LIN {X 0,Y 288.913,Z 1256.965,A -85,B 0,C 180,E1 22492.445,E2 22492.445} C_VEL
LIN {X 0,Y 288.678,Z 1266.037,A -85,B 0,C 180,E1 22499.979,E2 22499.979} C_VEL
LIN {X 0,Y 289.252,Z 1269.357,A -85,B 0,C 180,E1 22505.992,E2 22505.992} C_VEL
LIN {X 0,Y 291.406,Z 1269.606,A -85,B 0,C 180,E1 22511.982,E2 22511.982} C_VEL
LIN {X 0,Y 298.511,Z 1264.594,A -85,B 0,C 180,E1 22520.789,E2 22520.789} C_VEL
LIN {X 0,Y 311.662,Z 1253.252,A -85,B 0,C 180,E1 22529.064,E2 22529.064} C_VEL
LIN {X 0,Y 331.336,Z 1236.016,A -85,B 0,C 180,E1 22536.45,E2 22536.45} C_VEL
LIN {X 0,Y 358.761,Z 1211.96,A -85,B 0,C 180,E1 22542.945,E2 22542.945} C_VEL
LIN {X 0,Y 361.98,Z 1209.227,A -85,B 0,C 180,E1 22543.828,E2 22543.828} C_VEL
LIN {X 0,Y 332.745,Z 1238.454,A -85,B 0,C 180,E1 22549.983,E2 22549.983} C_VEL
LIN {X 0,Y 312.443,Z 1260.562,A -85,B 0,C 180,E1 22556.95,E2 22556.95} C_VEL
LIN {X 0,Y 299.017,Z 1276.755,A -85,B 0,C 180,E1 22564.501,E2 22564.501} C_VEL
LIN {X 0,Y 291.853,Z 1286.905,A -85,B 0,C 180,E1 22571.864,E2 22571.864} C_VEL
LIN {X 0,Y 289.278,Z 1291.684,A -85,B 0,C 180,E1 22577.92,E2 22577.92} C_VEL
LIN {X 0,Y 288.568,Z 1293.172,A -85,B 0,C 180,E1 22585.704,E2 22585.704} C_VEL
LIN {X 0,Y 288.992,Z 1290.468,A -85,B 0,C 180,E1 22591.516,E2 22591.516} C_VEL
LIN {X 0,Y 289.159,Z 1283.794,A -85,B 0,C 180,E1 22597.542,E2 22597.542} C_VEL
LIN {X 0,Y 290.047,Z 1270.937,A -85,B 0,C 180,E1 22604.382,E2 22604.382} C_VEL
LIN {X 0,Y 290.956,Z 1264.711,A -85,B 0,C 180,E1 22607.439,E2 22607.439} C_VEL
LIN {X 0,Y 296.193,Z 1251.831,A -85,B 0,C 180,E1 22614.979,E2 22614.979} C_VEL
LIN {X 0,Y 306.956,Z 1232.131,A -85,B 0,C 180,E1 22622.484,E2 22622.484} C_VEL
LIN {X 0,Y 322.211,Z 1206.964,A -85,B 0,C 180,E1 22628.94,E2 22628.94} C_VEL
LIN {X 0,Y 340.045,Z 1177.266,A -85,B 0,C 180,E1 22634.144,E2 22634.144} C_VEL
LIN {X 0,Y 358.723,Z 1143.523,A -85,B 0,C 180,E1 22638.132,E2 22638.132} C_VEL
LIN {X 0,Y 372.662,Z 1114.646,A -85,B 0,C 180,E1 22640.6,E2 22640.6} C_VEL
LIN {X 0,Y 373.421,Z 1108.193,A -85,B 0,C 180,E1 22642.533,E2 22642.533} C_VEL
LIN {X 0,Y 372.674,Z 1104.982,A -85,B 0,C 180,E1 22645.328,E2 22645.328} C_VEL
LIN {X 0,Y 372.153,Z 1105.867,A -85,B 0,C 180,E1 22648.785,E2 22648.785} C_VEL
LIN {X 0,Y 371.814,Z 1111.068,A -85,B 0,C 180,E1 22651.664,E2 22651.664} C_VEL
LIN {X 0,Y 356.252,Z 1142.151,A -85,B 0,C 180,E1 22654.514,E2 22654.514} C_VEL
LIN {X 0,Y 340.752,Z 1167.55,A -85,B 0,C 180,E1 22658.157,E2 22658.157} C_VEL
LIN {X 0,Y 330.737,Z 1181.649,A -85,B 0,C 180,E1 22661.066,E2 22661.066} C_VEL
LIN {X 0,Y 320.798,Z 1191.408,A -85,B 0,C 180,E1 22662.97,E2 22662.97} C_VEL
LIN {X 0,Y 312.043,Z 1198.825,A -85,B 0,C 180,E1 22664.79,E2 22664.79} C_VEL
LIN {X 0,Y 311.157,Z 1199.698,A -85,B 0,C 180,E1 22665.117,E2 22665.117} C_VEL
LIN {X 0,Y 298.817,Z 1210.613,A -85,B 0,C 180,E1 22671.272,E2 22671.272} C_VEL
LIN {X 0,Y 291.006,Z 1214.857,A -85,B 0,C 180,E1 22677.037,E2 22677.037} C_VEL
LIN {X 0,Y 285.807,Z 1214.307,A -85,B 0,C 180,E1 22683.06,E2 22683.06} C_VEL
LIN {X 0,Y 283.385,Z 1208.666,A -85,B 0,C 180,E1 22689.252,E2 22689.252} C_VEL
LIN {X 0,Y 283.421,Z 1196.875,A -85,B 0,C 180,E1 22695.723,E2 22695.723} C_VEL
LIN {X 0,Y 285.142,Z 1180.307,A -85,B 0,C 180,E1 22701.438,E2 22701.438} C_VEL
LIN {X 0,Y 288.359,Z 1157.155,A -85,B 0,C 180,E1 22706.832,E2 22706.832} C_VEL
LIN {X 0,Y 292.261,Z 1130.684,A -85,B 0,C 180,E1 22711.033,E2 22711.033} C_VEL
LIN {X 0,Y 296.144,Z 1100.075,A -85,B 0,C 180,E1 22714.272,E2 22714.272} C_VEL
LIN {X 0,Y 299.515,Z 1062.214,A -85,B 0,C 180,E1 22716.704,E2 22716.704} C_VEL
LIN {X 0,Y 299.117,Z 1052.067,A -85,B 0,C 180,E1 22717.323,E2 22717.323} C_VEL
LIN {X 0,Y 283.423,Z 996.5,A -85,B 0,C 180,E1 22721.746,E2 22721.746} C_VEL
LIN {X 0,Y 277.408,Z 977.53,A -85,B 0,C 180,E1 22723.544,E2 22723.544} C_VEL
LIN {X 0,Y 277.257,Z 977.53,A -85,B 0,C 180,E1 22733.028,E2 22733.028} C_VEL
LIN {X 0,Y 277.681,Z 977.53,A -85,B 0,C 180,E1 22740.854,E2 22740.854} C_VEL
LIN {X 0,Y 278.202,Z 977.53,A -85,B 0,C 180,E1 22747.851,E2 22747.851} C_VEL
LIN {X 0,Y 278.682,Z 977.53,A -85,B 0,C 180,E1 22754.21,E2 22754.21} C_VEL
LIN {X 0,Y 279.215,Z 977.53,A -85,B 0,C 180,E1 22760.616,E2 22760.616} C_VEL
LIN {X 0,Y 279.937,Z 977.53,A -85,B 0,C 180,E1 22766.883,E2 22766.883} C_VEL
LIN {X 0,Y 279.933,Z 977.53,A -85,B 0,C 180,E1 22773.088,E2 22773.088} C_VEL
LIN {X 0,Y 278.942,Z 977.53,A -85,B 0,C 180,E1 22782.535,E2 22782.535} C_VEL
LIN {X 0,Y 278.361,Z 977.53,A -85,B 0,C 180,E1 22789.048,E2 22789.048} C_VEL
LIN {X 0,Y 277.861,Z 977.53,A -85,B 0,C 180,E1 22795.85,E2 22795.85} C_VEL
LIN {X 0,Y 277.467,Z 977.53,A -85,B 0,C 180,E1 22804.97,E2 22804.97} C_VEL
LIN {X 0,Y 277.579,Z 977.96,A -85,B 0,C 180,E1 22805.92,E2 22805.92} C_VEL
LIN {X 0,Y 300.397,Z 1034.728,A -85,B 0,C 180,E1 22811.695,E2 22811.695} C_VEL
LIN {X 0,Y 313.014,Z 1073.998,A -85,B 0,C 180,E1 22815.793,E2 22815.793} C_VEL
LIN {X 0,Y 317.955,Z 1093.024,A -85,B 0,C 180,E1 22817.944,E2 22817.944} C_VEL
LIN {X 0,Y 309.265,Z 1133.148,A -85,B 0,C 180,E1 22821.776,E2 22821.776} C_VEL
LIN {X 0,Y 300.222,Z 1169.342,A -85,B 0,C 180,E1 22826.69,E2 22826.69} C_VEL
LIN {X 0,Y 292.592,Z 1198.797,A -85,B 0,C 180,E1 22832.199,E2 22832.199} C_VEL
LIN {X 0,Y 286.541,Z 1224.077,A -85,B 0,C 180,E1 22838.661,E2 22838.661} C_VEL
LIN {X 0,Y 282.581,Z 1244.505,A -85,B 0,C 180,E1 22846.016,E2 22846.016} C_VEL
LIN {X 0,Y 280.968,Z 1257.783,A -85,B 0,C 180,E1 22853.009,E2 22853.009} C_VEL
LIN {X 0,Y 280.777,Z 1266.014,A -85,B 0,C 180,E1 22859.978,E2 22859.978} C_VEL
LIN {X 0,Y 281.383,Z 1269.716,A -85,B 0,C 180,E1 22866.16,E2 22866.16} C_VEL
LIN {X 0,Y 283.679,Z 1270.268,A -85,B 0,C 180,E1 22872.313,E2 22872.313} C_VEL
LIN {X 0,Y 291.207,Z 1265.806,A -85,B 0,C 180,E1 22881.335,E2 22881.335} C_VEL
LIN {X 0,Y 305.036,Z 1255.326,A -85,B 0,C 180,E1 22889.758,E2 22889.758} C_VEL
LIN {X 0,Y 327.34,Z 1237.562,A -85,B 0,C 180,E1 22897.738,E2 22897.738} C_VEL
LIN {X 0,Y 352.425,Z 1217.519,A -85,B 0,C 180,E1 22903.435,E2 22903.435} C_VEL
LIN {X 0,Y 349.935,Z 1219.839,A -85,B 0,C 180,E1 22904.209,E2 22904.209} C_VEL
LIN {X 0,Y 319.79,Z 1247.985,A -85,B 0,C 180,E1 22911.126,E2 22911.126} C_VEL
LIN {X 0,Y 297.744,Z 1270.571,A -85,B 0,C 180,E1 22920,E2 22920} C_VEL
LIN {X 0,Y 286.72,Z 1283.669,A -85,B 0,C 180,E1 22928.303,E2 22928.303} C_VEL
LIN {X 0,Y 282.382,Z 1289.896,A -85,B 0,C 180,E1 22934.881,E2 22934.881} C_VEL
LIN {X 0,Y 280.916,Z 1292.547,A -85,B 0,C 180,E1 22940.702,E2 22940.702} C_VEL
LIN {X 0,Y 280.835,Z 1292.257,A -85,B 0,C 180,E1 22946.921,E2 22946.921} C_VEL
LIN {X 0,Y 281.131,Z 1289.623,A -85,B 0,C 180,E1 22951.559,E2 22951.559} C_VEL
LIN {X 0,Y 281.302,Z 1282.585,A -85,B 0,C 180,E1 22957.754,E2 22957.754} C_VEL
LIN {X 0,Y 282.209,Z 1270.064,A -85,B 0,C 180,E1 22964.483,E2 22964.483} C_VEL
LIN {X 0,Y 282.953,Z 1265.098,A -85,B 0,C 180,E1 22967.145,E2 22967.145} C_VEL
LIN {X 0,Y 288.891,Z 1251.656,A -85,B 0,C 180,E1 22975.656,E2 22975.656} C_VEL
LIN {X 0,Y 300.247,Z 1232.56,A -85,B 0,C 180,E1 22983.303,E2 22983.303} C_VEL
LIN {X 0,Y 316.13,Z 1208.273,A -85,B 0,C 180,E1 22989.817,E2 22989.817} C_VEL
LIN {X 0,Y 334.567,Z 1179.797,A -85,B 0,C 180,E1 22995.018,E2 22995.018} C_VEL
LIN {X 0,Y 353.854,Z 1147.351,A -85,B 0,C 180,E1 22999.019,E2 22999.019} C_VEL
LIN {X 0,Y 368.472,Z 1119.391,A -85,B 0,C 180,E1 23001.4,E2 23001.4} C_VEL
LIN {X 0,Y 369.311,Z 1113.908,A -85,B 0,C 180,E1 23003.254,E2 23003.254} C_VEL
LIN {X 0,Y 368.846,Z 1111.925,A -85,B 0,C 180,E1 23005.267,E2 23005.267} C_VEL
LIN {X 0,Y 368.267,Z 1112.965,A -85,B 0,C 180,E1 23008.847,E2 23008.847} C_VEL
LIN {X 0,Y 368.026,Z 1115.337,A -85,B 0,C 180,E1 23010.415,E2 23010.415} C_VEL
LIN {X 0,Y 366.892,Z 1118.227,A -85,B 0,C 180,E1 23010.936,E2 23010.936} C_VEL
LIN {X 0,Y 351.042,Z 1147.122,A -85,B 0,C 180,E1 23013.763,E2 23013.763} C_VEL
LIN {X 0,Y 335.04,Z 1171.219,A -85,B 0,C 180,E1 23017.415,E2 23017.415} C_VEL
LIN {X 0,Y 319.548,Z 1190.71,A -85,B 0,C 180,E1 23021.996,E2 23021.996} C_VEL
LIN {X 0,Y 311.157,Z 1199.698,A -85,B 0,C 180,E1 23025.117,E2 23025.117} C_VEL
LIN {X 0,Y 301.577,Z 1206.588,A -85,B 0,C 180,E1 23027.554,E2 23027.554} C_VEL
LIN {X 0,Y 293.227,Z 1211.363,A -85,B 0,C 180,E1 23029.856,E2 23029.856} C_VEL
LIN {X 0,Y 292.465,Z 1211.85,A -85,B 0,C 180,E1 23030.245,E2 23030.245} C_VEL
LIN {X 0,Y 283.133,Z 1216.283,A -85,B 0,C 180,E1 23036.954,E2 23036.954} C_VEL
LIN {X 0,Y 277.875,Z 1215.064,A -85,B 0,C 180,E1 23043.148,E2 23043.148} C_VEL
LIN {X 0,Y 275.444,Z 1208.736,A -85,B 0,C 180,E1 23049.521,E2 23049.521} C_VEL
LIN {X 0,Y 275.571,Z 1196.71,A -85,B 0,C 180,E1 23055.979,E2 23055.979} C_VEL
LIN {X 0,Y 277.478,Z 1179.1,A -85,B 0,C 180,E1 23061.994,E2 23061.994} C_VEL
LIN {X 0,Y 280.661,Z 1156.637,A -85,B 0,C 180,E1 23067.209,E2 23067.209} C_VEL
LIN {X 0,Y 284.645,Z 1130.244,A -85,B 0,C 180,E1 23071.454,E2 23071.454} C_VEL
LIN {X 0,Y 288.594,Z 1099.773,A -85,B 0,C 180,E1 23074.726,E2 23074.726} C_VEL
LIN {X 0,Y 292.242,Z 1059.083,A -85,B 0,C 180,E1 23077.358,E2 23077.358} C_VEL
LIN {X 0,Y 282.15,Z 1017.934,A -85,B 0,C 180,E1 23080.6,E2 23080.6} C_VEL
LIN {X 0,Y 269.397,Z 977.53,A -85,B 0,C 180,E1 23084.328,E2 23084.328} C_VEL
LIN {X 0,Y 269.242,Z 977.53,A -85,B 0,C 180,E1 23092.019,E2 23092.019} C_VEL
LIN {X 0,Y 269.549,Z 977.53,A -85,B 0,C 180,E1 23099.589,E2 23099.589} C_VEL
LIN {X 0,Y 270.123,Z 977.53,A -85,B 0,C 180,E1 23106.863,E2 23106.863} C_VEL
LIN {X 0,Y 270.679,Z 977.53,A -85,B 0,C 180,E1 23113.73,E2 23113.73} C_VEL
LIN {X 0,Y 271.289,Z 977.53,A -85,B 0,C 180,E1 23120.339,E2 23120.339} C_VEL
LIN {X 0,Y 272.024,Z 977.53,A -85,B 0,C 180,E1 23126.792,E2 23126.792} C_VEL
LIN {X 0,Y 272.019,Z 977.53,A -85,B 0,C 180,E1 23133.178,E2 23133.178} C_VEL
LIN {X 0,Y 271.263,Z 977.53,A -85,B 0,C 180,E1 23139.632,E2 23139.632} C_VEL
LIN {X 0,Y 270.47,Z 977.53,A -85,B 0,C 180,E1 23147.696,E2 23147.696} C_VEL
LIN {X 0,Y 269.94,Z 977.53,A -85,B 0,C 180,E1 23156.048,E2 23156.048} C_VEL
LIN {X 0,Y 269.572,Z 977.695,A -85,B 0,C 180,E1 23164.793,E2 23164.793} C_VEL
LIN {X 0,Y 292.525,Z 1034.517,A -85,B 0,C 180,E1 23170.823,E2 23170.823} C_VEL
LIN {X 0,Y 305.526,Z 1075.222,A -85,B 0,C 180,E1 23175.204,E2 23175.204} C_VEL
LIN {X 0,Y 310.377,Z 1095.235,A -85,B 0,C 180,E1 23177.517,E2 23177.517} C_VEL
LIN {X 0,Y 301.699,Z 1134.071,A -85,B 0,C 180,E1 23181.347,E2 23181.347} C_VEL
LIN {X 0,Y 292.601,Z 1169.644,A -85,B 0,C 180,E1 23186.3,E2 23186.3} C_VEL
LIN {X 0,Y 284.518,Z 1200.304,A -85,B 0,C 180,E1 23192.204,E2 23192.204} C_VEL
LIN {X 0,Y 278.158,Z 1226.524,A -85,B 0,C 180,E1 23199.241,E2 23199.241} C_VEL
LIN {X 0,Y 274.526,Z 1245.536,A -85,B 0,C 180,E1 23206.448,E2 23206.448} C_VEL
LIN {X 0,Y 273.004,Z 1258.55,A -85,B 0,C 180,E1 23213.605,E2 23213.605} C_VEL
LIN {X 0,Y 272.903,Z 1265.954,A -85,B 0,C 180,E1 23219.977,E2 23219.977} C_VEL
LIN {X 0,Y 273.53,Z 1270.023,A -85,B 0,C 180,E1 23226.337,E2 23226.337} C_VEL
LIN {X 0,Y 275.96,Z 1270.937,A -85,B 0,C 180,E1 23232.663,E2 23232.663} C_VEL
LIN {X 0,Y 283.929,Z 1267.034,A -85,B 0,C 180,E1 23241.91,E2 23241.91} C_VEL
LIN {X 0,Y 298.433,Z 1257.296,A -85,B 0,C 180,E1 23250.485,E2 23250.485} C_VEL
LIN {X 0,Y 321.645,Z 1240.685,A -85,B 0,C 180,E1 23258.527,E2 23258.527} C_VEL
LIN {X 0,Y 342.424,Z 1225.545,A -85,B 0,C 180,E1 23263.266,E2 23263.266} C_VEL
LIN {X 0,Y 343.123,Z 1225.113,A -85,B 0,C 180,E1 23263.689,E2 23263.689} C_VEL
LIN {X 0,Y 311.936,Z 1251.882,A -85,B 0,C 180,E1 23270.857,E2 23270.857} C_VEL
LIN {X 0,Y 289.855,Z 1272.711,A -85,B 0,C 180,E1 23279.817,E2 23279.817} C_VEL
LIN {X 0,Y 277.869,Z 1285.614,A -85,B 0,C 180,E1 23289.256,E2 23289.256} C_VEL
LIN {X 0,Y 273.627,Z 1291.227,A -85,B 0,C 180,E1 23297.218,E2 23297.218} C_VEL
LIN {X 0,Y 272.852,Z 1292.257,A -85,B 0,C 180,E1 23303.638,E2 23303.638} C_VEL
LIN {X 0,Y 273.451,Z 1289.888,A -85,B 0,C 180,E1 23310.015,E2 23310.015} C_VEL
LIN {X 0,Y 273.431,Z 1282.535,A -85,B 0,C 180,E1 23317.178,E2 23317.178} C_VEL
LIN {X 0,Y 274.227,Z 1270.393,A -85,B 0,C 180,E1 23324.035,E2 23324.035} C_VEL
LIN {X 0,Y 274.729,Z 1266.131,A -85,B 0,C 180,E1 23326.023,E2 23326.023} C_VEL
LIN {X 0,Y 279.954,Z 1254.348,A -85,B 0,C 180,E1 23334.817,E2 23334.817} C_VEL
LIN {X 0,Y 291.472,Z 1236.104,A -85,B 0,C 180,E1 23343.1,E2 23343.1} C_VEL
LIN {X 0,Y 308.835,Z 1211.543,A -85,B 0,C 180,E1 23350.298,E2 23350.298} C_VEL
LIN {X 0,Y 328.243,Z 1183.776,A -85,B 0,C 180,E1 23355.704,E2 23355.704} C_VEL
LIN {X 0,Y 348.455,Z 1152.244,A -85,B 0,C 180,E1 23359.81,E2 23359.81} C_VEL
LIN {X 0,Y 364.712,Z 1123.183,A -85,B 0,C 180,E1 23362.414,E2 23362.414} C_VEL
LIN {X 0,Y 364.999,Z 1119.391,A -85,B 0,C 180,E1 23364.491,E2 23364.491} C_VEL
LIN {X 0,Y 364.303,Z 1119.747,A -85,B 0,C 180,E1 23368.697,E2 23368.697} C_VEL
LIN {X 0,Y 364.117,Z 1120.792,A -85,B 0,C 180,E1 23369.482,E2 23369.482} C_VEL
LIN {X 0,Y 363.326,Z 1122.74,A -85,B 0,C 180,E1 23369.993,E2 23369.993} C_VEL
LIN {X 0,Y 347.159,Z 1150.07,A -85,B 0,C 180,E1 23372.746,E2 23372.746} C_VEL
LIN {X 0,Y 329.855,Z 1174.272,A -85,B 0,C 180,E1 23376.529,E2 23376.529} C_VEL
LIN {X 0,Y 314.156,Z 1192.562,A -85,B 0,C 180,E1 23380.985,E2 23380.985} C_VEL
LIN {X 0,Y 300.527,Z 1205.679,A -85,B 0,C 180,E1 23386.166,E2 23386.166} C_VEL
LIN {X 0,Y 292.465,Z 1211.85,A -85,B 0,C 180,E1 23390.245,E2 23390.245} C_VEL
LIN {X 0,Y 283.823,Z 1215.533,A -85,B 0,C 180,E1 23393.197,E2 23393.197} C_VEL
LIN {X 0,Y 275.941,Z 1217.538,A -85,B 0,C 180,E1 23396.245,E2 23396.245} C_VEL
LIN {X 0,Y 275.811,Z 1217.449,A -85,B 0,C 180,E1 23396.355,E2 23396.355} C_VEL
LIN {X 0,Y 269.9,Z 1215.69,A -85,B 0,C 180,E1 23403.241,E2 23403.241} C_VEL
LIN {X 0,Y 267.509,Z 1208.732,A -85,B 0,C 180,E1 23409.806,E2 23409.806} C_VEL
LIN {X 0,Y 267.753,Z 1195.931,A -85,B 0,C 180,E1 23416.459,E2 23416.459} C_VEL
LIN {X 0,Y 269.831,Z 1177.507,A -85,B 0,C 180,E1 23422.652,E2 23422.652} C_VEL
LIN {X 0,Y 273.347,Z 1153.731,A -85,B 0,C 180,E1 23428.069,E2 23428.069} C_VEL
LIN {X 0,Y 277.462,Z 1126.067,A -85,B 0,C 180,E1 23432.366,E2 23432.366} C_VEL
LIN {X 0,Y 281.463,Z 1095.674,A -85,B 0,C 180,E1 23435.502,E2 23435.502} C_VEL
LIN {X 0,Y 284.345,Z 1056.162,A -85,B 0,C 180,E1 23438.081,E2 23438.081} C_VEL
LIN {X 0,Y 269.556,Z 1002.727,A -85,B 0,C 180,E1 23442.632,E2 23442.632} C_VEL
LIN {X 0,Y 261.427,Z 977.53,A -85,B 0,C 180,E1 23445.044,E2 23445.044} C_VEL
LIN {X 0,Y 261.299,Z 977.53,A -85,B 0,C 180,E1 23454.538,E2 23454.538} C_VEL
LIN {X 0,Y 261.789,Z 977.53,A -85,B 0,C 180,E1 23462.399,E2 23462.399} C_VEL
LIN {X 0,Y 262.369,Z 977.53,A -85,B 0,C 180,E1 23469.709,E2 23469.709} C_VEL
LIN {X 0,Y 263.089,Z 977.53,A -85,B 0,C 180,E1 23478.353,E2 23478.353} C_VEL
LIN {X 0,Y 264.09,Z 977.53,A -85,B 0,C 180,E1 23486.695,E2 23486.695} C_VEL
LIN {X 0,Y 264.478,Z 977.53,A -85,B 0,C 180,E1 23489.985,E2 23489.985} C_VEL
LIN {X 0,Y 263.652,Z 977.53,A -85,B 0,C 180,E1 23496.585,E2 23496.585} C_VEL
LIN {X 0,Y 262.984,Z 977.53,A -85,B 0,C 180,E1 23503.309,E2 23503.309} C_VEL
LIN {X 0,Y 262.183,Z 977.53,A -85,B 0,C 180,E1 23512.331,E2 23512.331} C_VEL
LIN {X 0,Y 261.6,Z 977.53,A -85,B 0,C 180,E1 23521.402,E2 23521.402} C_VEL
LIN {X 0,Y 261.605,Z 977.53,A -85,B 0,C 180,E1 23523.583,E2 23523.583} C_VEL
LIN {X 0,Y 284.389,Z 1033.775,A -85,B 0,C 180,E1 23529.851,E2 23529.851} C_VEL
LIN {X 0,Y 297.241,Z 1073.785,A -85,B 0,C 180,E1 23534.297,E2 23534.297} C_VEL
LIN {X 0,Y 302.876,Z 1096.857,A -85,B 0,C 180,E1 23537.031,E2 23537.031} C_VEL
LIN {X 0,Y 293.687,Z 1136.512,A -85,B 0,C 180,E1 23541.092,E2 23541.092} C_VEL
LIN {X 0,Y 284.47,Z 1171.588,A -85,B 0,C 180,E1 23546.175,E2 23546.175} C_VEL
LIN {X 0,Y 276.388,Z 1201.702,A -85,B 0,C 180,E1 23552.203,E2 23552.203} C_VEL
LIN {X 0,Y 270.331,Z 1226.439,A -85,B 0,C 180,E1 23559.042,E2 23559.042} C_VEL
LIN {X 0,Y 266.477,Z 1246.367,A -85,B 0,C 180,E1 23566.831,E2 23566.831} C_VEL
LIN {X 0,Y 265.029,Z 1259.283,A -85,B 0,C 180,E1 23574.235,E2 23574.235} C_VEL
LIN {X 0,Y 265,Z 1267.449,A -85,B 0,C 180,E1 23581.779,E2 23581.779} C_VEL
LIN {X 0,Y 266.684,Z 1271.263,A -85,B 0,C 180,E1 23589.79,E2 23589.79} C_VEL
LIN {X 0,Y 273.176,Z 1270.019,A -85,B 0,C 180,E1 23599.49,E2 23599.49} C_VEL
LIN {X 0,Y 286.075,Z 1262.888,A -85,B 0,C 180,E1 23608.442,E2 23608.442} C_VEL
LIN {X 0,Y 307.827,Z 1249.109,A -85,B 0,C 180,E1 23617.055,E2 23617.055} C_VEL
LIN {X 0,Y 334.236,Z 1231.739,A -85,B 0,C 180,E1 23623.519,E2 23623.519} C_VEL
LIN {X 0,Y 304.547,Z 1255.198,A -85,B 0,C 180,E1 23630.416,E2 23630.416} C_VEL
LIN {X 0,Y 281.712,Z 1274.755,A -85,B 0,C 180,E1 23639.735,E2 23639.735} C_VEL
LIN {X 0,Y 270.386,Z 1285.758,A -85,B 0,C 180,E1 23648.654,E2 23648.654} C_VEL
LIN {X 0,Y 265.814,Z 1290.899,A -85,B 0,C 180,E1 23656.835,E2 23656.835} C_VEL
LIN {X 0,Y 264.965,Z 1291.615,A -85,B 0,C 180,E1 23663.448,E2 23663.448} C_VEL
LIN {X 0,Y 265.59,Z 1289.004,A -85,B 0,C 180,E1 23670.015,E2 23670.015} C_VEL
LIN {X 0,Y 265.618,Z 1282.453,A -85,B 0,C 180,E1 23676.567,E2 23676.567} C_VEL
LIN {X 0,Y 266.388,Z 1269.417,A -85,B 0,C 180,E1 23684.14,E2 23684.14} C_VEL
LIN {X 0,Y 266.951,Z 1265.43,A -85,B 0,C 180,E1 23686.503,E2 23686.503} C_VEL
LIN {X 0,Y 272.632,Z 1254.122,A -85,B 0,C 180,E1 23695.531,E2 23695.531} C_VEL
LIN {X 0,Y 284.723,Z 1236.648,A -85,B 0,C 180,E1 23703.928,E2 23703.928} C_VEL
LIN {X 0,Y 303.222,Z 1212.495,A -85,B 0,C 180,E1 23711.343,E2 23711.343} C_VEL
LIN {X 0,Y 324.201,Z 1184.531,A -85,B 0,C 180,E1 23716.929,E2 23716.929} C_VEL
LIN {X 0,Y 345.84,Z 1152.886,A -85,B 0,C 180,E1 23721.069,E2 23721.069} C_VEL
LIN {X 0,Y 360.586,Z 1128.204,A -85,B 0,C 180,E1 23723.275,E2 23723.275} C_VEL
LIN {X 0,Y 360.841,Z 1126.758,A -85,B 0,C 180,E1 23724.018,E2 23724.018} C_VEL
LIN {X 0,Y 360.377,Z 1125.639,A -85,B 0,C 180,E1 23727.259,E2 23727.259} C_VEL
LIN {X 0,Y 360.15,Z 1126.687,A -85,B 0,C 180,E1 23728.72,E2 23728.72} C_VEL
LIN {X 0,Y 358.221,Z 1130.165,A -85,B 0,C 180,E1 23729.274,E2 23729.274} C_VEL
LIN {X 0,Y 340.802,Z 1156.828,A -85,B 0,C 180,E1 23732.193,E2 23732.193} C_VEL
LIN {X 0,Y 323.141,Z 1179.261,A -85,B 0,C 180,E1 23736.011,E2 23736.011} C_VEL
LIN {X 0,Y 306.919,Z 1196.489,A -85,B 0,C 180,E1 23740.582,E2 23740.582} C_VEL
LIN {X 0,Y 291.59,Z 1209.561,A -85,B 0,C 180,E1 23746.5,E2 23746.5} C_VEL
LIN {X 0,Y 283.474,Z 1214.755,A -85,B 0,C 180,E1 23750.795,E2 23750.795} C_VEL
LIN {X 0,Y 275.811,Z 1217.449,A -85,B 0,C 180,E1 23756.355,E2 23756.355} C_VEL
LIN {X 0,Y 268.497,Z 1217.81,A -85,B 0,C 180,E1 23759.701,E2 23759.701} C_VEL
LIN {X 0,Y 262.016,Z 1216.329,A -85,B 0,C 180,E1 23763.206,E2 23763.206} C_VEL
LIN {X 0,Y 259.582,Z 1208.572,A -85,B 0,C 180,E1 23770.109,E2 23770.109} C_VEL
LIN {X 0,Y 259.908,Z 1195.113,A -85,B 0,C 180,E1 23776.971,E2 23776.971} C_VEL
LIN {X 0,Y 262.252,Z 1175.727,A -85,B 0,C 180,E1 23783.349,E2 23783.349} C_VEL
LIN {X 0,Y 265.933,Z 1151.784,A -85,B 0,C 180,E1 23788.739,E2 23788.739} C_VEL
LIN {X 0,Y 269.983,Z 1124.57,A -85,B 0,C 180,E1 23792.95,E2 23792.95} C_VEL
LIN {X 0,Y 274.246,Z 1092.367,A -85,B 0,C 180,E1 23796.216,E2 23796.216} C_VEL
LIN {X 0,Y 276.817,Z 1057.498,A -85,B 0,C 180,E1 23798.531,E2 23798.531} C_VEL
LIN {X 0,Y 261.766,Z 1003.117,A -85,B 0,C 180,E1 23803.348,E2 23803.348} C_VEL
LIN {X 0,Y 253.452,Z 977.53,A -85,B 0,C 180,E1 23805.993,E2 23805.993} C_VEL
LIN {X 0,Y 253.231,Z 977.53,A -85,B 0,C 180,E1 23813.227,E2 23813.227} C_VEL
LIN {X 0,Y 253.771,Z 977.53,A -85,B 0,C 180,E1 23821.448,E2 23821.448} C_VEL
LIN {X 0,Y 254.402,Z 977.53,A -85,B 0,C 180,E1 23829.044,E2 23829.044} C_VEL
LIN {X 0,Y 254.993,Z 977.53,A -85,B 0,C 180,E1 23836.233,E2 23836.233} C_VEL
LIN {X 0,Y 255.718,Z 977.53,A -85,B 0,C 180,E1 23843.178,E2 23843.178} C_VEL
LIN {X 0,Y 256.567,Z 977.53,A -85,B 0,C 180,E1 23849.984,E2 23849.984} C_VEL
LIN {X 0,Y 255.695,Z 977.53,A -85,B 0,C 180,E1 23856.791,E2 23856.791} C_VEL
LIN {X 0,Y 254.987,Z 977.53,A -85,B 0,C 180,E1 23863.735,E2 23863.735} C_VEL
LIN {X 0,Y 254.371,Z 977.53,A -85,B 0,C 180,E1 23870.924,E2 23870.924} C_VEL
LIN {X 0,Y 253.696,Z 977.53,A -85,B 0,C 180,E1 23880.692,E2 23880.692} C_VEL
LIN {X 0,Y 253.665,Z 977.557,A -85,B 0,C 180,E1 23882.388,E2 23882.388} C_VEL
LIN {X 0,Y 276.268,Z 1032.863,A -85,B 0,C 180,E1 23888.834,E2 23888.834} C_VEL
LIN {X 0,Y 288.914,Z 1071.81,A -85,B 0,C 180,E1 23893.295,E2 23893.295} C_VEL
LIN {X 0,Y 295.553,Z 1097.709,A -85,B 0,C 180,E1 23896.472,E2 23896.472} C_VEL
LIN {X 0,Y 285.937,Z 1138.05,A -85,B 0,C 180,E1 23900.735,E2 23900.735} C_VEL
LIN {X 0,Y 276.703,Z 1172.33,A -85,B 0,C 180,E1 23905.848,E2 23905.848} C_VEL
LIN {X 0,Y 268.256,Z 1203.166,A -85,B 0,C 180,E1 23912.235,E2 23912.235} C_VEL
LIN {X 0,Y 261.926,Z 1228.693,A -85,B 0,C 180,E1 23919.667,E2 23919.667} C_VEL
LIN {X 0,Y 258.445,Z 1247.235,A -85,B 0,C 180,E1 23927.276,E2 23927.276} C_VEL
LIN {X 0,Y 257.075,Z 1259.988,A -85,B 0,C 180,E1 23934.904,E2 23934.904} C_VEL
LIN {X 0,Y 257.112,Z 1267.219,A -85,B 0,C 180,E1 23941.664,E2 23941.664} C_VEL
LIN {X 0,Y 258.895,Z 1271.615,A -85,B 0,C 180,E1 23950.087,E2 23950.087} C_VEL
LIN {X 0,Y 265.679,Z 1271.021,A -85,B 0,C 180,E1 23959.984,E2 23959.984} C_VEL
LIN {X 0,Y 279.318,Z 1264.646,A -85,B 0,C 180,E1 23969.196,E2 23969.196} C_VEL
LIN {X 0,Y 301.933,Z 1251.806,A -85,B 0,C 180,E1 23977.904,E2 23977.904} C_VEL
LIN {X 0,Y 322.487,Z 1239.601,A -85,B 0,C 180,E1 23982.995,E2 23982.995} C_VEL
LIN {X 0,Y 323.737,Z 1238.966,A -85,B 0,C 180,E1 23983.618,E2 23983.618} C_VEL
LIN {X 0,Y 294.283,Z 1260.514,A -85,B 0,C 180,E1 23990.882,E2 23990.882} C_VEL
LIN {X 0,Y 272.956,Z 1277.216,A -85,B 0,C 180,E1 24000.042,E2 24000.042} C_VEL
LIN {X 0,Y 261.527,Z 1287.172,A -85,B 0,C 180,E1 24009.674,E2 24009.674} C_VEL
LIN {X 0,Y 257.31,Z 1291.142,A -85,B 0,C 180,E1 24019.84,E2 24019.84} C_VEL
LIN {X 0,Y 257.234,Z 1289.968,A -85,B 0,C 180,E1 24026.639,E2 24026.639} C_VEL
LIN {X 0,Y 257.593,Z 1286.56,A -85,B 0,C 180,E1 24031.87,E2 24031.87} C_VEL
LIN {X 0,Y 257.784,Z 1278.791,A -85,B 0,C 180,E1 24038.466,E2 24038.466} C_VEL
LIN {X 0,Y 258.891,Z 1265.808,A -85,B 0,C 180,E1 24045.566,E2 24045.566} C_VEL
LIN {X 0,Y 263.703,Z 1256.288,A -85,B 0,C 180,E1 24054.636,E2 24054.636} C_VEL
LIN {X 0,Y 275.363,Z 1240.507,A -85,B 0,C 180,E1 24063.404,E2 24063.404} C_VEL
LIN {X 0,Y 292.795,Z 1219.473,A -85,B 0,C 180,E1 24070.814,E2 24070.814} C_VEL
LIN {X 0,Y 314.25,Z 1193.22,A -85,B 0,C 180,E1 24076.847,E2 24076.847} C_VEL
LIN {X 0,Y 337.196,Z 1162.779,A -85,B 0,C 180,E1 24081.351,E2 24081.351} C_VEL
LIN {X 0,Y 355.622,Z 1134.856,A -85,B 0,C 180,E1 24084.073,E2 24084.073} C_VEL
LIN {X 0,Y 356.218,Z 1132.871,A -85,B 0,C 180,E1 24085.208,E2 24085.208} C_VEL
LIN {X 0,Y 356.035,Z 1132.551,A -85,B 0,C 180,E1 24087.589,E2 24087.589} C_VEL
LIN {X 0,Y 355.259,Z 1133.956,A -85,B 0,C 180,E1 24088.24,E2 24088.24} C_VEL
LIN {X 0,Y 335.7,Z 1161.585,A -85,B 0,C 180,E1 24091.366,E2 24091.366} C_VEL
LIN {X 0,Y 316.695,Z 1183.829,A -85,B 0,C 180,E1 24095.409,E2 24095.409} C_VEL
LIN {X 0,Y 299.81,Z 1200.078,A -85,B 0,C 180,E1 24100.103,E2 24100.103} C_VEL
LIN {X 0,Y 284.121,Z 1212.099,A -85,B 0,C 180,E1 24106.138,E2 24106.138} C_VEL
LIN {X 0,Y 275.789,Z 1216.714,A -85,B 0,C 180,E1 24110.537,E2 24110.537} C_VEL
LIN {X 0,Y 267.352,Z 1218.852,A -85,B 0,C 180,E1 24116.775,E2 24116.775} C_VEL
LIN {X 0,Y 262.016,Z 1216.329,A -85,B 0,C 180,E1 24123.206,E2 24123.206} C_VEL
LIN {X 0,Y 258.145,Z 1214.245,A -85,B 0,C 180,E1 24125.941,E2 24125.941} C_VEL
LIN {X 0,Y 251.793,Z 1209.077,A -85,B 0,C 180,E1 24130.003,E2 24130.003} C_VEL
LIN {X 0,Y 251.661,Z 1208.314,A -85,B 0,C 180,E1 24130.472,E2 24130.472} C_VEL
LIN {X 0,Y 252.178,Z 1194.061,A -85,B 0,C 180,E1 24137.507,E2 24137.507} C_VEL
LIN {X 0,Y 254.475,Z 1175.364,A -85,B 0,C 180,E1 24143.667,E2 24143.667} C_VEL
LIN {X 0,Y 258.319,Z 1150.931,A -85,B 0,C 180,E1 24149.207,E2 24149.207} C_VEL
LIN {X 0,Y 262.769,Z 1121.709,A -85,B 0,C 180,E1 24153.727,E2 24153.727} C_VEL
LIN {X 0,Y 266.996,Z 1089.736,A -85,B 0,C 180,E1 24156.892,E2 24156.892} C_VEL
LIN {X 0,Y 269.17,Z 1058.451,A -85,B 0,C 180,E1 24159.015,E2 24159.015} C_VEL
LIN {X 0,Y 254.281,Z 1004.344,A -85,B 0,C 180,E1 24164.021,E2 24164.021} C_VEL
LIN {X 0,Y 245.435,Z 977.53,A -85,B 0,C 180,E1 24166.831,E2 24166.831} C_VEL
LIN {X 0,Y 245.393,Z 977.53,A -85,B 0,C 180,E1 24176.219,E2 24176.219} C_VEL
LIN {X 0,Y 246.041,Z 977.53,A -85,B 0,C 180,E1 24184.444,E2 24184.444} C_VEL
LIN {X 0,Y 246.697,Z 977.53,A -85,B 0,C 180,E1 24192.098,E2 24192.098} C_VEL
LIN {X 0,Y 247.38,Z 977.53,A -85,B 0,C 180,E1 24199.395,E2 24199.395} C_VEL
LIN {X 0,Y 248.237,Z 977.53,A -85,B 0,C 180,E1 24206.484,E2 24206.484} C_VEL
LIN {X 0,Y 248.656,Z 977.53,A -85,B 0,C 180,E1 24209.984,E2 24209.984} C_VEL
LIN {X 0,Y 247.737,Z 977.53,A -85,B 0,C 180,E1 24217.01,E2 24217.01} C_VEL
LIN {X 0,Y 246.989,Z 977.53,A -85,B 0,C 180,E1 24224.188,E2 24224.188} C_VEL
LIN {X 0,Y 246.218,Z 977.53,A -85,B 0,C 180,E1 24232.564,E2 24232.564} C_VEL
LIN {X 0,Y 245.823,Z 977.634,A -85,B 0,C 180,E1 24241.131,E2 24241.131} C_VEL
LIN {X 0,Y 267.848,Z 1031.465,A -85,B 0,C 180,E1 24247.692,E2 24247.692} C_VEL
LIN {X 0,Y 281.037,Z 1071.51,A -85,B 0,C 180,E1 24252.45,E2 24252.45} C_VEL
LIN {X 0,Y 288.096,Z 1099.167,A -85,B 0,C 180,E1 24255.944,E2 24255.944} C_VEL
LIN {X 0,Y 278.434,Z 1138.521,A -85,B 0,C 180,E1 24260.226,E2 24260.226} C_VEL
LIN {X 0,Y 268.71,Z 1173.774,A -85,B 0,C 180,E1 24265.651,E2 24265.651} C_VEL
LIN {X 0,Y 260.16,Z 1204.272,A -85,B 0,C 180,E1 24272.205,E2 24272.205} C_VEL
LIN {X 0,Y 254.111,Z 1228.494,A -85,B 0,C 180,E1 24279.469,E2 24279.469} C_VEL
LIN {X 0,Y 250.668,Z 1246.352,A -85,B 0,C 180,E1 24286.874,E2 24286.874} C_VEL
LIN {X 0,Y 249.206,Z 1259.566,A -85,B 0,C 180,E1 24294.743,E2 24294.743} C_VEL
LIN {X 0,Y 249.216,Z 1267.094,A -85,B 0,C 180,E1 24301.717,E2 24301.717} C_VEL
LIN {X 0,Y 251.09,Z 1271.961,A -85,B 0,C 180,E1 24310.404,E2 24310.404} C_VEL
LIN {X 0,Y 258.291,Z 1271.927,A -85,B 0,C 180,E1 24320.581,E2 24320.581} C_VEL
LIN {X 0,Y 272.569,Z 1266.264,A -85,B 0,C 180,E1 24329.991,E2 24329.991} C_VEL
LIN {X 0,Y 296.122,Z 1254.536,A -85,B 0,C 180,E1 24338.785,E2 24338.785} C_VEL
LIN {X 0,Y 312.092,Z 1245.96,A -85,B 0,C 180,E1 24342.789,E2 24342.789} C_VEL
LIN {X 0,Y 313.742,Z 1245.221,A -85,B 0,C 180,E1 24343.596,E2 24343.596} C_VEL
LIN {X 0,Y 286.288,Z 1263.665,A -85,B 0,C 180,E1 24350.588,E2 24350.588} C_VEL
LIN {X 0,Y 266.084,Z 1277.927,A -85,B 0,C 180,E1 24359.186,E2 24359.186} C_VEL
LIN {X 0,Y 254.016,Z 1287.177,A -85,B 0,C 180,E1 24369.045,E2 24369.045} C_VEL
LIN {X 0,Y 249.452,Z 1290.629,A -85,B 0,C 180,E1 24379.517,E2 24379.517} C_VEL
LIN {X 0,Y 249.366,Z 1289.172,A -85,B 0,C 180,E1 24386.533,E2 24386.533} C_VEL
LIN {X 0,Y 249.773,Z 1285.507,A -85,B 0,C 180,E1 24391.928,E2 24391.928} C_VEL
LIN {X 0,Y 249.958,Z 1277.338,A -85,B 0,C 180,E1 24398.733,E2 24398.733} C_VEL
LIN {X 0,Y 251.038,Z 1265.272,A -85,B 0,C 180,E1 24405.595,E2 24405.595} C_VEL
LIN {X 0,Y 256.367,Z 1255.969,A -85,B 0,C 180,E1 24415.391,E2 24415.391} C_VEL
LIN {X 0,Y 269.77,Z 1239.621,A -85,B 0,C 180,E1 24424.903,E2 24424.903} C_VEL
LIN {X 0,Y 289.966,Z 1217.233,A -85,B 0,C 180,E1 24432.811,E2 24432.811} C_VEL
LIN {X 0,Y 312.885,Z 1191.083,A -85,B 0,C 180,E1 24438.666,E2 24438.666} C_VEL
LIN {X 0,Y 336.899,Z 1160.817,A -85,B 0,C 180,E1 24442.991,E2 24442.991} C_VEL
LIN {X 0,Y 351.488,Z 1139.97,A -85,B 0,C 180,E1 24445.014,E2 24445.014} C_VEL
LIN {X 0,Y 351.703,Z 1139.135,A -85,B 0,C 180,E1 24445.964,E2 24445.964} C_VEL
LIN {X 0,Y 351.077,Z 1139.842,A -85,B 0,C 180,E1 24447.375,E2 24447.375} C_VEL
LIN {X 0,Y 330.757,Z 1166.29,A -85,B 0,C 180,E1 24450.533,E2 24450.533} C_VEL
LIN {X 0,Y 310.001,Z 1188.469,A -85,B 0,C 180,E1 24454.841,E2 24454.841} C_VEL
LIN {X 0,Y 292.645,Z 1203.64,A -85,B 0,C 180,E1 24459.62,E2 24459.62} C_VEL
LIN {X 0,Y 276.632,Z 1214.56,A -85,B 0,C 180,E1 24465.755,E2 24465.755} C_VEL
LIN {X 0,Y 268.087,Z 1218.565,A -85,B 0,C 180,E1 24470.262,E2 24470.262} C_VEL
LIN {X 0,Y 259.435,Z 1219.964,A -85,B 0,C 180,E1 24476.676,E2 24476.676} C_VEL
LIN {X 0,Y 253.952,Z 1216.692,A -85,B 0,C 180,E1 24483.445,E2 24483.445} C_VEL
LIN {X 0,Y 251.661,Z 1208.314,A -85,B 0,C 180,E1 24490.472,E2 24490.472} C_VEL
LIN {X 0,Y 249.11,Z 1203.592,A -85,B 0,C 180,E1 24493.212,E2 24493.212} C_VEL
LIN {X 0,Y 244.317,Z 1195.045,A -85,B 0,C 180,E1 24497.238,E2 24497.238} C_VEL
LIN {X 0,Y 244.326,Z 1193.929,A -85,B 0,C 180,E1 24497.684,E2 24497.684} C_VEL
LIN {X 0,Y 246.819,Z 1174.203,A -85,B 0,C 180,E1 24504.197,E2 24504.197} C_VEL
LIN {X 0,Y 250.708,Z 1150.081,A -85,B 0,C 180,E1 24509.684,E2 24509.684} C_VEL
LIN {X 0,Y 255.148,Z 1121.484,A -85,B 0,C 180,E1 24514.162,E2 24514.162} C_VEL
LIN {X 0,Y 259.595,Z 1088.597,A -85,B 0,C 180,E1 24517.486,E2 24517.486} C_VEL
LIN {X 0,Y 261.731,Z 1060.341,A -85,B 0,C 180,E1 24519.445,E2 24519.445} C_VEL
LIN {X 0,Y 247.534,Z 1008.041,A -85,B 0,C 180,E1 24524.454,E2 24524.454} C_VEL
LIN {X 0,Y 237.427,Z 977.53,A -85,B 0,C 180,E1 24527.938,E2 24527.938} C_VEL
LIN {X 0,Y 237.5,Z 977.53,A -85,B 0,C 180,E1 24536.074,E2 24536.074} C_VEL
LIN {X 0,Y 237.939,Z 977.53,A -85,B 0,C 180,E1 24543.508,E2 24543.508} C_VEL
LIN {X 0,Y 238.792,Z 977.53,A -85,B 0,C 180,E1 24552.208,E2 24552.208} C_VEL
LIN {X 0,Y 239.426,Z 977.53,A -85,B 0,C 180,E1 24559.038,E2 24559.038} C_VEL
LIN {X 0,Y 240.307,Z 977.53,A -85,B 0,C 180,E1 24566.368,E2 24566.368} C_VEL
LIN {X 0,Y 240.745,Z 977.53,A -85,B 0,C 180,E1 24569.983,E2 24569.983} C_VEL
LIN {X 0,Y 239.794,Z 977.53,A -85,B 0,C 180,E1 24577.244,E2 24577.244} C_VEL
LIN {X 0,Y 238.981,Z 977.53,A -85,B 0,C 180,E1 24584.674,E2 24584.674} C_VEL
LIN {X 0,Y 238.352,Z 977.53,A -85,B 0,C 180,E1 24592.404,E2 24592.404} C_VEL
LIN {X 0,Y 237.888,Z 977.53,A -85,B 0,C 180,E1 24599.755,E2 24599.755} C_VEL
LIN {X 0,Y 259.741,Z 1030.687,A -85,B 0,C 180,E1 24606.574,E2 24606.574} C_VEL
LIN {X 0,Y 272.511,Z 1069.086,A -85,B 0,C 180,E1 24611.303,E2 24611.303} C_VEL
LIN {X 0,Y 280.651,Z 1100.476,A -85,B 0,C 180,E1 24615.397,E2 24615.397} C_VEL
LIN {X 0,Y 270.559,Z 1140.323,A -85,B 0,C 180,E1 24619.881,E2 24619.881} C_VEL
LIN {X 0,Y 260.681,Z 1175.219,A -85,B 0,C 180,E1 24625.453,E2 24625.453} C_VEL
LIN {X 0,Y 252.077,Z 1205.404,A -85,B 0,C 180,E1 24632.21,E2 24632.21} C_VEL
LIN {X 0,Y 246.025,Z 1229.45,A -85,B 0,C 180,E1 24639.706,E2 24639.706} C_VEL
LIN {X 0,Y 242.639,Z 1247.142,A -85,B 0,C 180,E1 24647.35,E2 24647.35} C_VEL
LIN {X 0,Y 241.26,Z 1260.212,A -85,B 0,C 180,E1 24655.472,E2 24655.472} C_VEL
LIN {X 0,Y 241.499,Z 1268.396,A -85,B 0,C 180,E1 24663.571,E2 24663.571} C_VEL
LIN {X 0,Y 243.303,Z 1272.297,A -85,B 0,C 180,E1 24670.741,E2 24670.741} C_VEL
LIN {X 0,Y 250.928,Z 1272.845,A -85,B 0,C 180,E1 24681.214,E2 24681.214} C_VEL
LIN {X 0,Y 265.883,Z 1267.904,A -85,B 0,C 180,E1 24690.827,E2 24690.827} C_VEL
LIN {X 0,Y 292.591,Z 1256.079,A -85,B 0,C 180,E1 24700.308,E2 24700.308} C_VEL
LIN {X 0,Y 304.713,Z 1250.282,A -85,B 0,C 180,E1 24703.239,E2 24703.239} C_VEL
LIN {X 0,Y 272.573,Z 1270.165,A -85,B 0,C 180,E1 24712.321,E2 24712.321} C_VEL
LIN {X 0,Y 254.216,Z 1282.063,A -85,B 0,C 180,E1 24721.539,E2 24721.539} C_VEL
LIN {X 0,Y 244.102,Z 1288.843,A -85,B 0,C 180,E1 24731.936,E2 24731.936} C_VEL
LIN {X 0,Y 241.627,Z 1290.073,A -85,B 0,C 180,E1 24739.173,E2 24739.173} C_VEL
LIN {X 0,Y 241.707,Z 1287.258,A -85,B 0,C 180,E1 24748.22,E2 24748.22} C_VEL
LIN {X 0,Y 242.077,Z 1280.776,A -85,B 0,C 180,E1 24755.404,E2 24755.404} C_VEL
LIN {X 0,Y 242.736,Z 1268.077,A -85,B 0,C 180,E1 24763.555,E2 24763.555} C_VEL
LIN {X 0,Y 243.161,Z 1264.686,A -85,B 0,C 180,E1 24765.568,E2 24765.568} C_VEL
LIN {X 0,Y 249.073,Z 1255.589,A -85,B 0,C 180,E1 24776.19,E2 24776.19} C_VEL
LIN {X 0,Y 262.125,Z 1241.14,A -85,B 0,C 180,E1 24785.334,E2 24785.334} C_VEL
LIN {X 0,Y 282.176,Z 1220.753,A -85,B 0,C 180,E1 24793.229,E2 24793.229} C_VEL
LIN {X 0,Y 305.365,Z 1196.343,A -85,B 0,C 180,E1 24799.196,E2 24799.196} C_VEL
LIN {X 0,Y 329.724,Z 1168.339,A -85,B 0,C 180,E1 24803.556,E2 24803.556} C_VEL
LIN {X 0,Y 345.638,Z 1147.62,A -85,B 0,C 180,E1 24805.73,E2 24805.73} C_VEL
LIN {X 0,Y 346.999,Z 1145.63,A -85,B 0,C 180,E1 24806.087,E2 24806.087} C_VEL
LIN {X 0,Y 346.183,Z 1146.587,A -85,B 0,C 180,E1 24806.588,E2 24806.588} C_VEL
LIN {X 0,Y 324.486,Z 1172.366,A -85,B 0,C 180,E1 24809.905,E2 24809.905} C_VEL
LIN {X 0,Y 303.034,Z 1193.219,A -85,B 0,C 180,E1 24814.307,E2 24814.307} C_VEL
LIN {X 0,Y 283.345,Z 1208.528,A -85,B 0,C 180,E1 24819.792,E2 24819.792} C_VEL
LIN {X 0,Y 269.136,Z 1216.922,A -85,B 0,C 180,E1 24825.349,E2 24825.349} C_VEL
LIN {X 0,Y 260.384,Z 1220.361,A -85,B 0,C 180,E1 24829.971,E2 24829.971} C_VEL
LIN {X 0,Y 251.521,Z 1221.034,A -85,B 0,C 180,E1 24836.571,E2 24836.571} C_VEL
LIN {X 0,Y 245.958,Z 1217.045,A -85,B 0,C 180,E1 24843.557,E2 24843.557} C_VEL
LIN {X 0,Y 243.758,Z 1208.001,A -85,B 0,C 180,E1 24850.772,E2 24850.772} C_VEL
LIN {X 0,Y 244.326,Z 1193.929,A -85,B 0,C 180,E1 24857.684,E2 24857.684} C_VEL
LIN {X 0,Y 241.466,Z 1184.655,A -85,B 0,C 180,E1 24861.122,E2 24861.122} C_VEL
LIN {X 0,Y 238.997,Z 1174.068,A -85,B 0,C 180,E1 24864.435,E2 24864.435} C_VEL
LIN {X 0,Y 243.127,Z 1149.205,A -85,B 0,C 180,E1 24870.19,E2 24870.19} C_VEL
LIN {X 0,Y 247.678,Z 1120.268,A -85,B 0,C 180,E1 24874.74,E2 24874.74} C_VEL
LIN {X 0,Y 252.081,Z 1087.982,A -85,B 0,C 180,E1 24878.029,E2 24878.029} C_VEL
LIN {X 0,Y 253.959,Z 1060.84,A -85,B 0,C 180,E1 24880.023,E2 24880.023} C_VEL
LIN {X 0,Y 240.207,Z 1009.902,A -85,B 0,C 180,E1 24885.088,E2 24885.088} C_VEL
LIN {X 0,Y 229.431,Z 977.53,A -85,B 0,C 180,E1 24888.903,E2 24888.903} C_VEL
LIN {X 0,Y 229.725,Z 977.53,A -85,B 0,C 180,E1 24899.076,E2 24899.076} C_VEL
LIN {X 0,Y 230.386,Z 977.53,A -85,B 0,C 180,E1 24907.095,E2 24907.095} C_VEL
LIN {X 0,Y 231.013,Z 977.53,A -85,B 0,C 180,E1 24914.771,E2 24914.771} C_VEL
LIN {X 0,Y 231.847,Z 977.53,A -85,B 0,C 180,E1 24922.472,E2 24922.472} C_VEL
LIN {X 0,Y 232.832,Z 977.53,A -85,B 0,C 180,E1 24929.983,E2 24929.983} C_VEL
LIN {X 0,Y 231.825,Z 977.53,A -85,B 0,C 180,E1 24937.494,E2 24937.494} C_VEL
LIN {X 0,Y 230.997,Z 977.53,A -85,B 0,C 180,E1 24945.194,E2 24945.194} C_VEL
LIN {X 0,Y 230.273,Z 977.53,A -85,B 0,C 180,E1 24953.236,E2 24953.236} C_VEL
LIN {X 0,Y 229.987,Z 977.901,A -85,B 0,C 180,E1 24958.36,E2 24958.36} C_VEL
LIN {X 0,Y 251.662,Z 1029.754,A -85,B 0,C 180,E1 24965.397,E2 24965.397} C_VEL
LIN {X 0,Y 264.179,Z 1067.416,A -85,B 0,C 180,E1 24970.19,E2 24970.19} C_VEL
LIN {X 0,Y 273.184,Z 1101.914,A -85,B 0,C 180,E1 24974.846,E2 24974.846} C_VEL
LIN {X 0,Y 262.803,Z 1141.492,A -85,B 0,C 180,E1 24979.447,E2 24979.447} C_VEL
LIN {X 0,Y 252.669,Z 1176.596,A -85,B 0,C 180,E1 24985.244,E2 24985.244} C_VEL
LIN {X 0,Y 243.967,Z 1206.468,A -85,B 0,C 180,E1 24992.211,E2 24992.211} C_VEL
LIN {X 0,Y 237.873,Z 1230.337,A -85,B 0,C 180,E1 24999.952,E2 24999.952} C_VEL
LIN {X 0,Y 234.615,Z 1247.882,A -85,B 0,C 180,E1 25007.858,E2 25007.858} C_VEL
LIN {X 0,Y 233.327,Z 1260.826,A -85,B 0,C 180,E1 25016.25,E2 25016.25} C_VEL
LIN {X 0,Y 233.609,Z 1268.226,A -85,B 0,C 180,E1 25023.692,E2 25023.692} C_VEL
LIN {X 0,Y 237.428,Z 1273.547,A -85,B 0,C 180,E1 25034.761,E2 25034.761} C_VEL
LIN {X 0,Y 247.982,Z 1272.893,A -85,B 0,C 180,E1 25045.293,E2 25045.293} C_VEL
LIN {X 0,Y 266.196,Z 1267.074,A -85,B 0,C 180,E1 25054.663,E2 25054.663} C_VEL
LIN {X 0,Y 294.693,Z 1255.49,A -85,B 0,C 180,E1 25063.351,E2 25063.351} C_VEL
LIN {X 0,Y 268.349,Z 1270.238,A -85,B 0,C 180,E1 25070.582,E2 25070.582} C_VEL
LIN {X 0,Y 247.189,Z 1282.379,A -85,B 0,C 180,E1 25080.652,E2 25080.652} C_VEL
LIN {X 0,Y 236.489,Z 1288.509,A -85,B 0,C 180,E1 25091.333,E2 25091.333} C_VEL
LIN {X 0,Y 233.499,Z 1288.727,A -85,B 0,C 180,E1 25102.56,E2 25102.56} C_VEL
LIN {X 0,Y 234.223,Z 1284.925,A -85,B 0,C 180,E1 25110.017,E2 25110.017} C_VEL
LIN {X 0,Y 234.287,Z 1277.034,A -85,B 0,C 180,E1 25117.449,E2 25117.449} C_VEL
LIN {X 0,Y 235.234,Z 1264.223,A -85,B 0,C 180,E1 25125.06,E2 25125.06} C_VEL
LIN {X 0,Y 239.729,Z 1257.584,A -85,B 0,C 180,E1 25134.777,E2 25134.777} C_VEL
LIN {X 0,Y 252.61,Z 1244.379,A -85,B 0,C 180,E1 25144.759,E2 25144.759} C_VEL
LIN {X 0,Y 272.262,Z 1225.927,A -85,B 0,C 180,E1 25153.002,E2 25153.002} C_VEL
LIN {X 0,Y 296.597,Z 1202.554,A -85,B 0,C 180,E1 25159.479,E2 25159.479} C_VEL
LIN {X 0,Y 322.553,Z 1175.274,A -85,B 0,C 180,E1 25164.152,E2 25164.152} C_VEL
LIN {X 0,Y 335.996,Z 1159.561,A -85,B 0,C 180,E1 25166.012,E2 25166.012} C_VEL
LIN {X 0,Y 337.08,Z 1158.127,A -85,B 0,C 180,E1 25166.343,E2 25166.343} C_VEL
LIN {X 0,Y 314.731,Z 1181.598,A -85,B 0,C 180,E1 25169.863,E2 25169.863} C_VEL
LIN {X 0,Y 292.581,Z 1200.477,A -85,B 0,C 180,E1 25174.568,E2 25174.568} C_VEL
LIN {X 0,Y 272.442,Z 1213.847,A -85,B 0,C 180,E1 25180.533,E2 25180.533} C_VEL
LIN {X 0,Y 258.443,Z 1220.385,A -85,B 0,C 180,E1 25186.463,E2 25186.463} C_VEL
LIN {X 0,Y 247.723,Z 1222.531,A -85,B 0,C 180,E1 25192.999,E2 25192.999} C_VEL
LIN {X 0,Y 240.37,Z 1220.221,A -85,B 0,C 180,E1 25200.026,E2 25200.026} C_VEL
LIN {X 0,Y 236.252,Z 1211.834,A -85,B 0,C 180,E1 25208.323,E2 25208.323} C_VEL
LIN {X 0,Y 236.128,Z 1197.932,A -85,B 0,C 180,E1 25216.09,E2 25216.09} C_VEL
LIN {X 0,Y 238.337,Z 1178.471,A -85,B 0,C 180,E1 25223.167,E2 25223.167} C_VEL
LIN {X 0,Y 238.997,Z 1174.068,A -85,B 0,C 180,E1 25224.435,E2 25224.435} C_VEL
LIN {X 0,Y 236.851,Z 1162.402,A -85,B 0,C 180,E1 25227.536,E2 25227.536} C_VEL
LIN {X 0,Y 235.024,Z 1151.272,A -85,B 0,C 180,E1 25230.1,E2 25230.1} C_VEL
LIN {X 0,Y 235.268,Z 1149.567,A -85,B 0,C 180,E1 25230.442,E2 25230.442} C_VEL
LIN {X 0,Y 240.043,Z 1120.258,A -85,B 0,C 180,E1 25235.197,E2 25235.197} C_VEL
LIN {X 0,Y 244.542,Z 1087.773,A -85,B 0,C 180,E1 25238.568,E2 25238.568} C_VEL
LIN {X 0,Y 246.422,Z 1062.342,A -85,B 0,C 180,E1 25240.5,E2 25240.5} C_VEL
LIN {X 0,Y 233.011,Z 1012.177,A -85,B 0,C 180,E1 25245.718,E2 25245.718} C_VEL
LIN {X 0,Y 221.492,Z 977.53,A -85,B 0,C 180,E1 25249.963,E2 25249.963} C_VEL
LIN {X 0,Y 221.46,Z 977.53,A -85,B 0,C 180,E1 25256.791,E2 25256.791} C_VEL
LIN {X 0,Y 222.198,Z 977.53,A -85,B 0,C 180,E1 25265.828,E2 25265.828} C_VEL
LIN {X 0,Y 222.986,Z 977.53,A -85,B 0,C 180,E1 25274.209,E2 25274.209} C_VEL
LIN {X 0,Y 223.898,Z 977.53,A -85,B 0,C 180,E1 25282.203,E2 25282.203} C_VEL
LIN {X 0,Y 224.926,Z 977.53,A -85,B 0,C 180,E1 25289.982,E2 25289.982} C_VEL
LIN {X 0,Y 223.876,Z 977.53,A -85,B 0,C 180,E1 25297.762,E2 25297.762} C_VEL
LIN {X 0,Y 222.749,Z 977.53,A -85,B 0,C 180,E1 25307.687,E2 25307.687} C_VEL
LIN {X 0,Y 222.067,Z 977.558,A -85,B 0,C 180,E1 25316.805,E2 25316.805} C_VEL
LIN {X 0,Y 244.103,Z 1030.197,A -85,B 0,C 180,E1 25324.347,E2 25324.347} C_VEL
LIN {X 0,Y 257.073,Z 1069.687,A -85,B 0,C 180,E1 25329.572,E2 25329.572} C_VEL
LIN {X 0,Y 265.636,Z 1103.576,A -85,B 0,C 180,E1 25334.309,E2 25334.309} C_VEL
LIN {X 0,Y 255.172,Z 1142.387,A -85,B 0,C 180,E1 25338.963,E2 25338.963} C_VEL
LIN {X 0,Y 244.7,Z 1177.836,A -85,B 0,C 180,E1 25345.029,E2 25345.029} C_VEL
LIN {X 0,Y 235.831,Z 1207.463,A -85,B 0,C 180,E1 25352.21,E2 25352.21} C_VEL
LIN {X 0,Y 229.749,Z 1231.163,A -85,B 0,C 180,E1 25360.218,E2 25360.218} C_VEL
LIN {X 0,Y 226.578,Z 1248.569,A -85,B 0,C 180,E1 25368.4,E2 25368.4} C_VEL
LIN {X 0,Y 225.412,Z 1261.401,A -85,B 0,C 180,E1 25377.083,E2 25377.083} C_VEL
LIN {X 0,Y 225.984,Z 1269.473,A -85,B 0,C 180,E1 25385.744,E2 25385.744} C_VEL
LIN {X 0,Y 229.785,Z 1273.879,A -85,B 0,C 180,E1 25395.264,E2 25395.264} C_VEL
LIN {X 0,Y 240.884,Z 1273.865,A -85,B 0,C 180,E1 25406.093,E2 25406.093} C_VEL
LIN {X 0,Y 263.864,Z 1267.6,A -85,B 0,C 180,E1 25417.049,E2 25417.049} C_VEL
LIN {X 0,Y 283.37,Z 1260.605,A -85,B 0,C 180,E1 25422.749,E2 25422.749} C_VEL
LIN {X 0,Y 284.064,Z 1260.461,A -85,B 0,C 180,E1 25423.431,E2 25423.431} C_VEL
LIN {X 0,Y 256.428,Z 1274.489,A -85,B 0,C 180,E1 25431.671,E2 25431.671} C_VEL
LIN {X 0,Y 237.774,Z 1283.983,A -85,B 0,C 180,E1 25441.468,E2 25441.468} C_VEL
LIN {X 0,Y 228.886,Z 1288.171,A -85,B 0,C 180,E1 25450.689,E2 25450.689} C_VEL
LIN {X 0,Y 225.647,Z 1287.88,A -85,B 0,C 180,E1 25462.3,E2 25462.3} C_VEL
LIN {X 0,Y 226.393,Z 1283.803,A -85,B 0,C 180,E1 25470.018,E2 25470.018} C_VEL
LIN {X 0,Y 226.462,Z 1275.446,A -85,B 0,C 180,E1 25477.708,E2 25477.708} C_VEL
LIN {X 0,Y 227.427,Z 1263.251,A -85,B 0,C 180,E1 25485.475,E2 25485.475} C_VEL
LIN {X 0,Y 231.997,Z 1257.436,A -85,B 0,C 180,E1 25495.141,E2 25495.141} C_VEL
LIN {X 0,Y 244.54,Z 1245.847,A -85,B 0,C 180,E1 25504.991,E2 25504.991} C_VEL
LIN {X 0,Y 266.371,Z 1227.116,A -85,B 0,C 180,E1 25514.097,E2 25514.097} C_VEL
LIN {X 0,Y 293.037,Z 1203.439,A -85,B 0,C 180,E1 25520.884,E2 25520.884} C_VEL
LIN {X 0,Y 319.814,Z 1177.235,A -85,B 0,C 180,E1 25525.428,E2 25525.428} C_VEL
LIN {X 0,Y 325.66,Z 1170.902,A -85,B 0,C 180,E1 25526.409,E2 25526.409} C_VEL
LIN {X 0,Y 302.189,Z 1192.145,A -85,B 0,C 180,E1 25530.347,E2 25530.347} C_VEL
LIN {X 0,Y 280.539,Z 1207.922,A -85,B 0,C 180,E1 25535.281,E2 25535.281} C_VEL
LIN {X 0,Y 261.341,Z 1218.48,A -85,B 0,C 180,E1 25541.431,E2 25541.431} C_VEL
LIN {X 0,Y 244.922,Z 1223.576,A -85,B 0,C 180,E1 25549.331,E2 25549.331} C_VEL
LIN {X 0,Y 235.648,Z 1222.79,A -85,B 0,C 180,E1 25556.34,E2 25556.34} C_VEL
LIN {X 0,Y 229.374,Z 1215.931,A -85,B 0,C 180,E1 25565.178,E2 25565.178} C_VEL
LIN {X 0,Y 227.973,Z 1203.424,A -85,B 0,C 180,E1 25573.478,E2 25573.478} C_VEL
LIN {X 0,Y 229.535,Z 1185.4,A -85,B 0,C 180,E1 25581.095,E2 25581.095} C_VEL
LIN {X 0,Y 233.083,Z 1162.199,A -85,B 0,C 180,E1 25587.711,E2 25587.711} C_VEL
LIN {X 0,Y 235.268,Z 1149.567,A -85,B 0,C 180,E1 25590.442,E2 25590.442} C_VEL
LIN {X 0,Y 234.587,Z 1139.329,A -85,B 0,C 180,E1 25592.45,E2 25592.45} C_VEL
LIN {X 0,Y 231.923,Z 1123.253,A -85,B 0,C 180,E1 25595.238,E2 25595.238} C_VEL
LIN {X 0,Y 232.158,Z 1121.331,A -85,B 0,C 180,E1 25595.506,E2 25595.506} C_VEL
LIN {X 0,Y 236.77,Z 1090.08,A -85,B 0,C 180,E1 25598.929,E2 25598.929} C_VEL
LIN {X 0,Y 239.012,Z 1064.227,A -85,B 0,C 180,E1 25600.965,E2 25600.965} C_VEL
LIN {X 0,Y 226.066,Z 1015.109,A -85,B 0,C 180,E1 25606.288,E2 25606.288} C_VEL
LIN {X 0,Y 213.515,Z 977.53,A -85,B 0,C 180,E1 25611.072,E2 25611.072} C_VEL
LIN {X 0,Y 213.722,Z 977.53,A -85,B 0,C 180,E1 25620.223,E2 25620.223} C_VEL
LIN {X 0,Y 214.552,Z 977.53,A -85,B 0,C 180,E1 25629.302,E2 25629.302} C_VEL
LIN {X 0,Y 215.422,Z 977.53,A -85,B 0,C 180,E1 25637.799,E2 25637.799} C_VEL
LIN {X 0,Y 216.457,Z 977.53,A -85,B 0,C 180,E1 25645.967,E2 25645.967} C_VEL
LIN {X 0,Y 217.009,Z 977.53,A -85,B 0,C 180,E1 25649.981,E2 25649.981} C_VEL
LIN {X 0,Y 215.893,Z 977.53,A -85,B 0,C 180,E1 25658.05,E2 25658.05} C_VEL
LIN {X 0,Y 214.968,Z 977.53,A -85,B 0,C 180,E1 25666.357,E2 25666.357} C_VEL
LIN {X 0,Y 214.208,Z 977.533,A -85,B 0,C 180,E1 25675.195,E2 25675.195} C_VEL
LIN {X 0,Y 235.714,Z 1028.769,A -85,B 0,C 180,E1 25682.964,E2 25682.964} C_VEL
LIN {X 0,Y 248.712,Z 1067.804,A -85,B 0,C 180,E1 25688.344,E2 25688.344} C_VEL
LIN {X 0,Y 258.051,Z 1103.534,A -85,B 0,C 180,E1 25693.532,E2 25693.532} C_VEL
LIN {X 0,Y 247.854,Z 1142.147,A -85,B 0,C 180,E1 25698.302,E2 25698.302} C_VEL
LIN {X 0,Y 237.04,Z 1177.922,A -85,B 0,C 180,E1 25704.57,E2 25704.57} C_VEL
LIN {X 0,Y 228.194,Z 1206.796,A -85,B 0,C 180,E1 25711.736,E2 25711.736} C_VEL
LIN {X 0,Y 221.915,Z 1230.738,A -85,B 0,C 180,E1 25720.01,E2 25720.01} C_VEL
LIN {X 0,Y 218.542,Z 1249.21,A -85,B 0,C 180,E1 25728.98,E2 25728.98} C_VEL
LIN {X 0,Y 217.558,Z 1261.94,A -85,B 0,C 180,E1 25737.976,E2 25737.976} C_VEL
LIN {X 0,Y 218.536,Z 1270.645,A -85,B 0,C 180,E1 25747.942,E2 25747.942} C_VEL
LIN {X 0,Y 225.091,Z 1275.017,A -85,B 0,C 180,E1 25759.638,E2 25759.638} C_VEL
LIN {X 0,Y 239.584,Z 1273.939,A -85,B 0,C 180,E1 25770.361,E2 25770.361} C_VEL
LIN {X 0,Y 266.487,Z 1266.839,A -85,B 0,C 180,E1 25780.8,E2 25780.8} C_VEL
LIN {X 0,Y 274.195,Z 1264.389,A -85,B 0,C 180,E1 25782.891,E2 25782.891} C_VEL
LIN {X 0,Y 272.53,Z 1265.292,A -85,B 0,C 180,E1 25783.736,E2 25783.736} C_VEL
LIN {X 0,Y 242.732,Z 1278.823,A -85,B 0,C 180,E1 25793.648,E2 25793.648} C_VEL
LIN {X 0,Y 224.31,Z 1286.805,A -85,B 0,C 180,E1 25806.109,E2 25806.109} C_VEL
LIN {X 0,Y 218.199,Z 1287.993,A -85,B 0,C 180,E1 25817.994,E2 25817.994} C_VEL
LIN {X 0,Y 218.228,Z 1283.958,A -85,B 0,C 180,E1 25828.029,E2 25828.029} C_VEL
LIN {X 0,Y 218.637,Z 1277.636,A -85,B 0,C 180,E1 25834.988,E2 25834.988} C_VEL
LIN {X 0,Y 219.288,Z 1265.045,A -85,B 0,C 180,E1 25843.53,E2 25843.53} C_VEL
LIN {X 0,Y 219.554,Z 1262.446,A -85,B 0,C 180,E1 25845.069,E2 25845.069} C_VEL
LIN {X 0,Y 224.69,Z 1256.856,A -85,B 0,C 180,E1 25856.018,E2 25856.018} C_VEL
LIN {X 0,Y 239.555,Z 1244.638,A -85,B 0,C 180,E1 25866.956,E2 25866.956} C_VEL
LIN {X 0,Y 262.853,Z 1226.451,A -85,B 0,C 180,E1 25875.924,E2 25875.924} C_VEL
LIN {X 0,Y 289.672,Z 1204.44,A -85,B 0,C 180,E1 25882.319,E2 25882.319} C_VEL
LIN {X 0,Y 313.149,Z 1183.131,A -85,B 0,C 180,E1 25886.169,E2 25886.169} C_VEL
LIN {X 0,Y 313.436,Z 1182.742,A -85,B 0,C 180,E1 25886.607,E2 25886.607} C_VEL
LIN {X 0,Y 288.978,Z 1201.736,A -85,B 0,C 180,E1 25891.014,E2 25891.014} C_VEL
LIN {X 0,Y 266.646,Z 1215.216,A -85,B 0,C 180,E1 25896.588,E2 25896.588} C_VEL
LIN {X 0,Y 250.188,Z 1222.266,A -85,B 0,C 180,E1 25902.401,E2 25902.401} C_VEL
LIN {X 0,Y 237.182,Z 1225.033,A -85,B 0,C 180,E1 25908.978,E2 25908.978} C_VEL
LIN {X 0,Y 227.705,Z 1223.52,A -85,B 0,C 180,E1 25916.212,E2 25916.212} C_VEL
LIN {X 0,Y 221.456,Z 1216.003,A -85,B 0,C 180,E1 25925.194,E2 25925.194} C_VEL
LIN {X 0,Y 220.107,Z 1202.919,A -85,B 0,C 180,E1 25933.736,E2 25933.736} C_VEL
LIN {X 0,Y 221.706,Z 1185.115,A -85,B 0,C 180,E1 25941.312,E2 25941.312} C_VEL
LIN {X 0,Y 225.345,Z 1161.714,A -85,B 0,C 180,E1 25948.107,E2 25948.107} C_VEL
LIN {X 0,Y 230.142,Z 1134.195,A -85,B 0,C 180,E1 25953.572,E2 25953.572} C_VEL
LIN {X 0,Y 232.158,Z 1121.331,A -85,B 0,C 180,E1 25955.506,E2 25955.506} C_VEL
LIN {X 0,Y 232.157,Z 1113.699,A -85,B 0,C 180,E1 25956.574,E2 25956.574} C_VEL
LIN {X 0,Y 228.925,Z 1092.309,A -85,B 0,C 180,E1 25959.289,E2 25959.289} C_VEL
LIN {X 0,Y 229.171,Z 1090.243,A -85,B 0,C 180,E1 25959.473,E2 25959.473} C_VEL
LIN {X 0,Y 231.332,Z 1065.047,A -85,B 0,C 180,E1 25961.576,E2 25961.576} C_VEL
LIN {X 0,Y 218.741,Z 1017.043,A -85,B 0,C 180,E1 25966.983,E2 25966.983} C_VEL
LIN {X 0,Y 205.519,Z 977.53,A -85,B 0,C 180,E1 25972.317,E2 25972.317} C_VEL
LIN {X 0,Y 205.863,Z 977.53,A -85,B 0,C 180,E1 25982.09,E2 25982.09} C_VEL
LIN {X 0,Y 206.537,Z 977.53,A -85,B 0,C 180,E1 25988.459,E2 25988.459} C_VEL
LIN {X 0,Y 207.403,Z 977.53,A -85,B 0,C 180,E1 25997.319,E2 25997.319} C_VEL
LIN {X 0,Y 208.499,Z 977.53,A -85,B 0,C 180,E1 26005.813,E2 26005.813} C_VEL
LIN {X 0,Y 209.112,Z 977.53,A -85,B 0,C 180,E1 26009.981,E2 26009.981} C_VEL
LIN {X 0,Y 207.936,Z 977.53,A -85,B 0,C 180,E1 26018.361,E2 26018.361} C_VEL
LIN {X 0,Y 206.814,Z 977.53,A -85,B 0,C 180,E1 26027.659,E2 26027.659} C_VEL
LIN {X 0,Y 206.379,Z 977.936,A -85,B 0,C 180,E1 26033.511,E2 26033.511} C_VEL
LIN {X 0,Y 226.983,Z 1026.109,A -85,B 0,C 180,E1 26041.347,E2 26041.347} C_VEL
LIN {X 0,Y 240.392,Z 1065.719,A -85,B 0,C 180,E1 26047.042,E2 26047.042} C_VEL
LIN {X 0,Y 250.205,Z 1103.535,A -85,B 0,C 180,E1 26052.697,E2 26052.697} C_VEL
LIN {X 0,Y 249.649,Z 1110.056,A -85,B 0,C 180,E1 26053.527,E2 26053.527} C_VEL
LIN {X 0,Y 238.436,Z 1149.063,A -85,B 0,C 180,E1 26058.722,E2 26058.722} C_VEL
LIN {X 0,Y 227.719,Z 1183.062,A -85,B 0,C 180,E1 26065.238,E2 26065.238} C_VEL
LIN {X 0,Y 219.023,Z 1211.29,A -85,B 0,C 180,E1 26072.859,E2 26072.859} C_VEL
LIN {X 0,Y 213.256,Z 1233.827,A -85,B 0,C 180,E1 26081.324,E2 26081.324} C_VEL
LIN {X 0,Y 210.387,Z 1251.495,A -85,B 0,C 180,E1 26090.645,E2 26090.645} C_VEL
LIN {X 0,Y 209.784,Z 1263.523,A -85,B 0,C 180,E1 26099.97,E2 26099.97} C_VEL
LIN {X 0,Y 211.341,Z 1271.68,A -85,B 0,C 180,E1 26110.295,E2 26110.295} C_VEL
LIN {X 0,Y 217.629,Z 1275.48,A -85,B 0,C 180,E1 26120.34,E2 26120.34} C_VEL
LIN {X 0,Y 232.861,Z 1275.094,A -85,B 0,C 180,E1 26131.335,E2 26131.335} C_VEL
LIN {X 0,Y 260.79,Z 1268.995,A -85,B 0,C 180,E1 26141.889,E2 26141.889} C_VEL
LIN {X 0,Y 263.157,Z 1268.316,A -85,B 0,C 180,E1 26142.538,E2 26142.538} C_VEL
LIN {X 0,Y 263.95,Z 1268.245,A -85,B 0,C 180,E1 26143.335,E2 26143.335} C_VEL
LIN {X 0,Y 232.833,Z 1280.766,A -85,B 0,C 180,E1 26154.168,E2 26154.168} C_VEL
LIN {X 0,Y 217.013,Z 1286.494,A -85,B 0,C 180,E1 26165.253,E2 26165.253} C_VEL
LIN {X 0,Y 210.426,Z 1287.125,A -85,B 0,C 180,E1 26177.544,E2 26177.544} C_VEL
LIN {X 0,Y 210.414,Z 1282.78,A -85,B 0,C 180,E1 26187.956,E2 26187.956} C_VEL
LIN {X 0,Y 210.845,Z 1276.143,A -85,B 0,C 180,E1 26195.173,E2 26195.173} C_VEL
LIN {X 0,Y 211.666,Z 1262.184,A -85,B 0,C 180,E1 26204.516,E2 26204.516} C_VEL
LIN {X 0,Y 219.368,Z 1254.717,A -85,B 0,C 180,E1 26218.936,E2 26218.936} C_VEL
LIN {X 0,Y 237.128,Z 1241.999,A -85,B 0,C 180,E1 26229.981,E2 26229.981} C_VEL
LIN {X 0,Y 262.69,Z 1223.672,A -85,B 0,C 180,E1 26238.602,E2 26238.602} C_VEL
LIN {X 0,Y 290.83,Z 1202.001,A -85,B 0,C 180,E1 26244.521,E2 26244.521} C_VEL
LIN {X 0,Y 302.532,Z 1192.099,A -85,B 0,C 180,E1 26246.597,E2 26246.597} C_VEL
LIN {X 0,Y 277.194,Z 1209.083,A -85,B 0,C 180,E1 26251.386,E2 26251.386} C_VEL
LIN {X 0,Y 256.534,Z 1219.597,A -85,B 0,C 180,E1 26256.85,E2 26256.85} C_VEL
LIN {X 0,Y 242.786,Z 1224.374,A -85,B 0,C 180,E1 26261.846,E2 26261.846} C_VEL
LIN {X 0,Y 229.436,Z 1226.35,A -85,B 0,C 180,E1 26268.601,E2 26268.601} C_VEL
LIN {X 0,Y 219.742,Z 1224.099,A -85,B 0,C 180,E1 26276.075,E2 26276.075} C_VEL
LIN {X 0,Y 213.631,Z 1216.319,A -85,B 0,C 180,E1 26284.945,E2 26284.945} C_VEL
LIN {X 0,Y 212.196,Z 1203.762,A -85,B 0,C 180,E1 26293.25,E2 26293.25} C_VEL
LIN {X 0,Y 213.557,Z 1186.78,A -85,B 0,C 180,E1 26300.808,E2 26300.808} C_VEL
LIN {X 0,Y 216.892,Z 1164.807,A -85,B 0,C 180,E1 26307.599,E2 26307.599} C_VEL
LIN {X 0,Y 221.596,Z 1138.859,A -85,B 0,C 180,E1 26313.193,E2 26313.193} C_VEL
LIN {X 0,Y 226.849,Z 1107.391,A -85,B 0,C 180,E1 26317.735,E2 26317.735} C_VEL
LIN {X 0,Y 229.171,Z 1090.243,A -85,B 0,C 180,E1 26319.473,E2 26319.473} C_VEL
LIN {X 0,Y 228.272,Z 1078.049,A -85,B 0,C 180,E1 26320.684,E2 26320.684} C_VEL
LIN {X 0,Y 221.945,Z 1058.383,A -85,B 0,C 180,E1 26323.011,E2 26323.011} C_VEL
LIN {X 0,Y 209.614,Z 1012.637,A -85,B 0,C 180,E1 26328.53,E2 26328.53} C_VEL
LIN {X 0,Y 197.562,Z 977.53,A -85,B 0,C 180,E1 26333.656,E2 26333.656} C_VEL
LIN {X 0,Y 198.024,Z 977.53,A -85,B 0,C 180,E1 26342.647,E2 26342.647} C_VEL
LIN {X 0,Y 198.919,Z 977.53,A -85,B 0,C 180,E1 26352.239,E2 26352.239} C_VEL
LIN {X 0,Y 199.955,Z 977.53,A -85,B 0,C 180,E1 26361.262,E2 26361.262} C_VEL
LIN {X 0,Y 201.19,Z 977.53,A -85,B 0,C 180,E1 26369.98,E2 26369.98} C_VEL
LIN {X 0,Y 199.775,Z 977.53,A -85,B 0,C 180,E1 26379.441,E2 26379.441} C_VEL
LIN {X 0,Y 198.652,Z 977.53,A -85,B 0,C 180,E1 26390.053,E2 26390.053} C_VEL
LIN {X 0,Y 198.624,Z 977.794,A -85,B 0,C 180,E1 26391.664,E2 26391.664} C_VEL
LIN {X 0,Y 219.019,Z 1025.658,A -85,B 0,C 180,E1 26399.94,E2 26399.94} C_VEL
LIN {X 0,Y 231.652,Z 1062.245,A -85,B 0,C 180,E1 26405.466,E2 26405.466} C_VEL
LIN {X 0,Y 241.491,Z 1099.59,A -85,B 0,C 180,E1 26411.208,E2 26411.208} C_VEL
LIN {X 0,Y 242.697,Z 1109.213,A -85,B 0,C 180,E1 26412.67,E2 26412.67} C_VEL
LIN {X 0,Y 231.038,Z 1148.905,A -85,B 0,C 180,E1 26418.046,E2 26418.046} C_VEL
LIN {X 0,Y 220.049,Z 1182.951,A -85,B 0,C 180,E1 26424.751,E2 26424.751} C_VEL
LIN {X 0,Y 211.038,Z 1211.583,A -85,B 0,C 180,E1 26432.73,E2 26432.73} C_VEL
LIN {X 0,Y 205.145,Z 1234.474,A -85,B 0,C 180,E1 26441.675,E2 26441.675} C_VEL
LIN {X 0,Y 202.364,Z 1252.021,A -85,B 0,C 180,E1 26451.357,E2 26451.357} C_VEL
LIN {X 0,Y 201.933,Z 1263.971,A -85,B 0,C 180,E1 26461.044,E2 26461.044} C_VEL
LIN {X 0,Y 203.55,Z 1271.58,A -85,B 0,C 180,E1 26470.693,E2 26470.693} C_VEL
LIN {X 0,Y 210.203,Z 1275.794,A -85,B 0,C 180,E1 26481.092,E2 26481.092} C_VEL
LIN {X 0,Y 226.193,Z 1276.125,A -85,B 0,C 180,E1 26492.369,E2 26492.369} C_VEL
LIN {X 0,Y 254.032,Z 1271.237,A -85,B 0,C 180,E1 26502.727,E2 26502.727} C_VEL
LIN {X 0,Y 251.952,Z 1272.143,A -85,B 0,C 180,E1 26503.829,E2 26503.829} C_VEL
LIN {X 0,Y 223.885,Z 1281.971,A -85,B 0,C 180,E1 26514.251,E2 26514.251} C_VEL
LIN {X 0,Y 209.742,Z 1286.179,A -85,B 0,C 180,E1 26524.334,E2 26524.334} C_VEL
LIN {X 0,Y 202.676,Z 1286.22,A -85,B 0,C 180,E1 26537.059,E2 26537.059} C_VEL
LIN {X 0,Y 202.641,Z 1281.457,A -85,B 0,C 180,E1 26547.877,E2 26547.877} C_VEL
LIN {X 0,Y 203.074,Z 1274.476,A -85,B 0,C 180,E1 26555.372,E2 26555.372} C_VEL
LIN {X 0,Y 203.906,Z 1260.261,A -85,B 0,C 180,E1 26565.113,E2 26565.113} C_VEL
LIN {X 0,Y 210.238,Z 1255.52,A -85,B 0,C 180,E1 26577.957,E2 26577.957} C_VEL
LIN {X 0,Y 226.691,Z 1244.903,A -85,B 0,C 180,E1 26589.304,E2 26589.304} C_VEL
LIN {X 0,Y 252.89,Z 1228.03,A -85,B 0,C 180,E1 26598.687,E2 26598.687} C_VEL
LIN {X 0,Y 283.53,Z 1206.546,A -85,B 0,C 180,E1 26605.279,E2 26605.279} C_VEL
LIN {X 0,Y 290.949,Z 1200.928,A -85,B 0,C 180,E1 26606.462,E2 26606.462} C_VEL
LIN {X 0,Y 262.508,Z 1216.863,A -85,B 0,C 180,E1 26612.528,E2 26612.528} C_VEL
LIN {X 0,Y 243.591,Z 1224.26,A -85,B 0,C 180,E1 26618.115,E2 26618.115} C_VEL
LIN {X 0,Y 228.066,Z 1227.495,A -85,B 0,C 180,E1 26624.618,E2 26624.618} C_VEL
LIN {X 0,Y 216.221,Z 1226.635,A -85,B 0,C 180,E1 26631.973,E2 26631.973} C_VEL
LIN {X 0,Y 207.631,Z 1220.426,A -85,B 0,C 180,E1 26641.075,E2 26641.075} C_VEL
LIN {X 0,Y 204.427,Z 1209.767,A -85,B 0,C 180,E1 26649.63,E2 26649.63} C_VEL
LIN {X 0,Y 204.995,Z 1193.037,A -85,B 0,C 180,E1 26658.339,E2 26658.339} C_VEL
LIN {X 0,Y 207.965,Z 1171.58,A -85,B 0,C 180,E1 26665.953,E2 26665.953} C_VEL
LIN {X 0,Y 212.795,Z 1145.105,A -85,B 0,C 180,E1 26672.401,E2 26672.401} C_VEL
LIN {X 0,Y 218.106,Z 1114.373,A -85,B 0,C 180,E1 26677.412,E2 26677.412} C_VEL
LIN {X 0,Y 222.846,Z 1079.631,A -85,B 0,C 180,E1 26680.972,E2 26680.972} C_VEL
LIN {X 0,Y 223.722,Z 1066.188,A -85,B 0,C 180,E1 26682.138,E2 26682.138} C_VEL
LIN {X 0,Y 221.945,Z 1058.383,A -85,B 0,C 180,E1 26683.011,E2 26683.011} C_VEL
LIN {X 0,Y 216.947,Z 1047.642,A -85,B 0,C 180,E1 26684.494,E2 26684.494} C_VEL
LIN {X 0,Y 207.718,Z 1032.526,A -85,B 0,C 180,E1 26686.959,E2 26686.959} C_VEL
LIN {X 0,Y 207.106,Z 1030.618,A -85,B 0,C 180,E1 26687.216,E2 26687.216} C_VEL
LIN {X 0,Y 193.719,Z 989.336,A -85,B 0,C 180,E1 26693.024,E2 26693.024} C_VEL
LIN {X 0,Y 189.634,Z 977.53,A -85,B 0,C 180,E1 26694.931,E2 26694.931} C_VEL
LIN {X 0,Y 190.394,Z 977.53,A -85,B 0,C 180,E1 26706.528,E2 26706.528} C_VEL
LIN {X 0,Y 191.334,Z 977.53,A -85,B 0,C 180,E1 26716.234,E2 26716.234} C_VEL
LIN {X 0,Y 192.584,Z 977.53,A -85,B 0,C 180,E1 26725.466,E2 26725.466} C_VEL
LIN {X 0,Y 193.265,Z 977.53,A -85,B 0,C 180,E1 26729.979,E2 26729.979} C_VEL
LIN {X 0,Y 191.948,Z 977.53,A -85,B 0,C 180,E1 26739.063,E2 26739.063} C_VEL
LIN {X 0,Y 190.778,Z 977.863,A -85,B 0,C 180,E1 26749.655,E2 26749.655} C_VEL
LIN {X 0,Y 211.005,Z 1024.672,A -85,B 0,C 180,E1 26758.387,E2 26758.387} C_VEL
LIN {X 0,Y 223.797,Z 1061.634,A -85,B 0,C 180,E1 26764.229,E2 26764.229} C_VEL
LIN {X 0,Y 233.494,Z 1098.385,A -85,B 0,C 180,E1 26770.105,E2 26770.105} C_VEL
LIN {X 0,Y 235.574,Z 1109.037,A -85,B 0,C 180,E1 26771.852,E2 26771.852} C_VEL
LIN {X 0,Y 223.688,Z 1148.623,A -85,B 0,C 180,E1 26777.328,E2 26777.328} C_VEL
LIN {X 0,Y 212.397,Z 1182.768,A -85,B 0,C 180,E1 26784.229,E2 26784.229} C_VEL
LIN {X 0,Y 203.419,Z 1210.719,A -85,B 0,C 180,E1 26792.223,E2 26792.223} C_VEL
LIN {X 0,Y 197.293,Z 1233.866,A -85,B 0,C 180,E1 26801.499,E2 26801.499} C_VEL
LIN {X 0,Y 194.55,Z 1250.827,A -85,B 0,C 180,E1 26811.007,E2 26811.007} C_VEL
LIN {X 0,Y 194.07,Z 1263.313,A -85,B 0,C 180,E1 26821.086,E2 26821.086} C_VEL
LIN {X 0,Y 196.773,Z 1272.581,A -85,B 0,C 180,E1 26833.323,E2 26833.323} C_VEL
LIN {X 0,Y 207.409,Z 1276.979,A -85,B 0,C 180,E1 26845.961,E2 26845.961} C_VEL
LIN {X 0,Y 227.083,Z 1276.519,A -85,B 0,C 180,E1 26856.87,E2 26856.87} C_VEL
LIN {X 0,Y 244.713,Z 1273.847,A -85,B 0,C 180,E1 26862.89,E2 26862.89} C_VEL
LIN {X 0,Y 213.169,Z 1283.345,A -85,B 0,C 180,E1 26875.366,E2 26875.366} C_VEL
LIN {X 0,Y 198.879,Z 1286.25,A -85,B 0,C 180,E1 26887.629,E2 26887.629} C_VEL
LIN {X 0,Y 194.362,Z 1283.819,A -85,B 0,C 180,E1 26901.051,E2 26901.051} C_VEL
LIN {X 0,Y 195.257,Z 1278.429,A -85,B 0,C 180,E1 26910.021,E2 26910.021} C_VEL
LIN {X 0,Y 195.28,Z 1269.982,A -85,B 0,C 180,E1 26917.825,E2 26917.825} C_VEL
LIN {X 0,Y 196.144,Z 1258.944,A -85,B 0,C 180,E1 26925.283,E2 26925.283} C_VEL
LIN {X 0,Y 201.163,Z 1255.87,A -85,B 0,C 180,E1 26936.891,E2 26936.891} C_VEL
LIN {X 0,Y 217.127,Z 1246.856,A -85,B 0,C 180,E1 26948.933,E2 26948.933} C_VEL
LIN {X 0,Y 242.518,Z 1232.171,A -85,B 0,C 180,E1 26958.595,E2 26958.595} C_VEL
LIN {X 0,Y 271.924,Z 1213.672,A -85,B 0,C 180,E1 26965.304,E2 26965.304} C_VEL
LIN {X 0,Y 278.734,Z 1209.045,A -85,B 0,C 180,E1 26966.469,E2 26966.469} C_VEL
LIN {X 0,Y 278.104,Z 1209.236,A -85,B 0,C 180,E1 26967.016,E2 26967.016} C_VEL
LIN {X 0,Y 253.093,Z 1221.084,A -85,B 0,C 180,E1 26972.386,E2 26972.386} C_VEL
LIN {X 0,Y 236.387,Z 1226.529,A -85,B 0,C 180,E1 26977.412,E2 26977.412} C_VEL
LIN {X 0,Y 220.475,Z 1228.96,A -85,B 0,C 180,E1 26984.075,E2 26984.075} C_VEL
LIN {X 0,Y 208.325,Z 1227.336,A -85,B 0,C 180,E1 26991.667,E2 26991.667} C_VEL
LIN {X 0,Y 199.592,Z 1220.316,A -85,B 0,C 180,E1 27001.118,E2 27001.118} C_VEL
LIN {X 0,Y 196.485,Z 1208.873,A -85,B 0,C 180,E1 27010.023,E2 27010.023} C_VEL
LIN {X 0,Y 197.151,Z 1192.652,A -85,B 0,C 180,E1 27018.515,E2 27018.515} C_VEL
LIN {X 0,Y 200.293,Z 1170.27,A -85,B 0,C 180,E1 27026.529,E2 27026.529} C_VEL
LIN {X 0,Y 205.241,Z 1143.876,A -85,B 0,C 180,E1 27033.021,E2 27033.021} C_VEL
LIN {X 0,Y 210.713,Z 1113.097,A -85,B 0,C 180,E1 27038.114,E2 27038.114} C_VEL
LIN {X 0,Y 215.622,Z 1077.518,A -85,B 0,C 180,E1 27041.802,E2 27041.802} C_VEL
LIN {X 0,Y 215.968,Z 1066.597,A -85,B 0,C 180,E1 27042.823,E2 27042.823} C_VEL
LIN {X 0,Y 207.106,Z 1030.618,A -85,B 0,C 180,E1 27047.216,E2 27047.216} C_VEL
LIN {X 0,Y 201.615,Z 1020.314,A -85,B 0,C 180,E1 27048.912,E2 27048.912} C_VEL
LIN {X 0,Y 191.796,Z 1005.932,A -85,B 0,C 180,E1 27051.74,E2 27051.74} C_VEL
LIN {X 0,Y 191.111,Z 1004.073,A -85,B 0,C 180,E1 27052.032,E2 27052.032} C_VEL
LIN {X 0,Y 181.657,Z 977.53,A -85,B 0,C 180,E1 27056.578,E2 27056.578} C_VEL
LIN {X 0,Y 182.393,Z 977.53,A -85,B 0,C 180,E1 27066.111,E2 27066.111} C_VEL
LIN {X 0,Y 183.314,Z 977.53,A -85,B 0,C 180,E1 27075.619,E2 27075.619} C_VEL
LIN {X 0,Y 184.611,Z 977.53,A -85,B 0,C 180,E1 27085.27,E2 27085.27} C_VEL
LIN {X 0,Y 185.337,Z 977.53,A -85,B 0,C 180,E1 27089.978,E2 27089.978} C_VEL
LIN {X 0,Y 183.947,Z 977.53,A -85,B 0,C 180,E1 27099.46,E2 27099.46} C_VEL
LIN {X 0,Y 183.099,Z 977.715,A -85,B 0,C 180,E1 27107.509,E2 27107.509} C_VEL
LIN {X 0,Y 202.436,Z 1022.562,A -85,B 0,C 180,E1 27116.499,E2 27116.499} C_VEL
LIN {X 0,Y 215.036,Z 1058.551,A -85,B 0,C 180,E1 27122.493,E2 27122.493} C_VEL
LIN {X 0,Y 225.075,Z 1095.325,A -85,B 0,C 180,E1 27128.62,E2 27128.62} C_VEL
LIN {X 0,Y 227.975,Z 1110.614,A -85,B 0,C 180,E1 27131.2,E2 27131.2} C_VEL
LIN {X 0,Y 215.533,Z 1150.729,A -85,B 0,C 180,E1 27137.011,E2 27137.011} C_VEL
LIN {X 0,Y 204.133,Z 1184.393,A -85,B 0,C 180,E1 27144.145,E2 27144.145} C_VEL
LIN {X 0,Y 194.756,Z 1213.172,A -85,B 0,C 180,E1 27152.876,E2 27152.876} C_VEL
LIN {X 0,Y 188.728,Z 1236.837,A -85,B 0,C 180,E1 27163.113,E2 27163.113} C_VEL
LIN {X 0,Y 186.397,Z 1252.91,A -85,B 0,C 180,E1 27172.963,E2 27172.963} C_VEL
LIN {X 0,Y 186.356,Z 1264.732,A -85,B 0,C 180,E1 27183.462,E2 27183.462} C_VEL
LIN {X 0,Y 190.269,Z 1273.538,A -85,B 0,C 180,E1 27196.149,E2 27196.149} C_VEL
LIN {X 0,Y 200.32,Z 1277.38,A -85,B 0,C 180,E1 27206.953,E2 27206.953} C_VEL
LIN {X 0,Y 220.855,Z 1277.599,A -85,B 0,C 180,E1 27218.091,E2 27218.091} C_VEL
LIN {X 0,Y 233.756,Z 1276.277,A -85,B 0,C 180,E1 27222.575,E2 27222.575} C_VEL
LIN {X 0,Y 233.238,Z 1276.59,A -85,B 0,C 180,E1 27223.408,E2 27223.408} C_VEL
LIN {X 0,Y 206.628,Z 1283.32,A -85,B 0,C 180,E1 27234.104,E2 27234.104} C_VEL
LIN {X 0,Y 191.513,Z 1285.501,A -85,B 0,C 180,E1 27246.719,E2 27246.719} C_VEL
LIN {X 0,Y 186.605,Z 1282.564,A -85,B 0,C 180,E1 27260.676,E2 27260.676} C_VEL
LIN {X 0,Y 187.532,Z 1276.829,A -85,B 0,C 180,E1 27270.022,E2 27270.022} C_VEL
LIN {X 0,Y 187.518,Z 1268.024,A -85,B 0,C 180,E1 27278.151,E2 27278.151} C_VEL
LIN {X 0,Y 188.374,Z 1257.558,A -85,B 0,C 180,E1 27285.295,E2 27285.295} C_VEL
LIN {X 0,Y 193.975,Z 1254.981,A -85,B 0,C 180,E1 27297.973,E2 27297.973} C_VEL
LIN {X 0,Y 210.907,Z 1246.627,A -85,B 0,C 180,E1 27310.311,E2 27310.311} C_VEL
LIN {X 0,Y 237.357,Z 1232.913,A -85,B 0,C 180,E1 27320.028,E2 27320.028} C_VEL
LIN {X 0,Y 266.126,Z 1216.349,A -85,B 0,C 180,E1 27326.394,E2 27326.394} C_VEL
LIN {X 0,Y 267.137,Z 1215.588,A -85,B 0,C 180,E1 27326.983,E2 27326.983} C_VEL
LIN {X 0,Y 243.675,Z 1224.871,A -85,B 0,C 180,E1 27332.233,E2 27332.233} C_VEL
LIN {X 0,Y 220.561,Z 1229.964,A -85,B 0,C 180,E1 27339.942,E2 27339.942} C_VEL
LIN {X 0,Y 206.14,Z 1229.61,A -85,B 0,C 180,E1 27347.293,E2 27347.293} C_VEL
LIN {X 0,Y 195.806,Z 1225.125,A -85,B 0,C 180,E1 27355.594,E2 27355.594} C_VEL
LIN {X 0,Y 189.507,Z 1214.651,A -85,B 0,C 180,E1 27365.768,E2 27365.768} C_VEL
LIN {X 0,Y 188.722,Z 1198.128,A -85,B 0,C 180,E1 27375.868,E2 27375.868} C_VEL
LIN {X 0,Y 191.142,Z 1178.115,A -85,B 0,C 180,E1 27384.162,E2 27384.162} C_VEL
LIN {X 0,Y 195.813,Z 1152.031,A -85,B 0,C 180,E1 27391.617,E2 27391.617} C_VEL
LIN {X 0,Y 201.249,Z 1122.677,A -85,B 0,C 180,E1 27397.28,E2 27397.28} C_VEL
LIN {X 0,Y 206.602,Z 1089.926,A -85,B 0,C 180,E1 27401.34,E2 27401.34} C_VEL
LIN {X 0,Y 208.569,Z 1068.501,A -85,B 0,C 180,E1 27403.378,E2 27403.378} C_VEL
LIN {X 0,Y 196.894,Z 1022.238,A -85,B 0,C 180,E1 27409.368,E2 27409.368} C_VEL
LIN {X 0,Y 191.111,Z 1004.073,A -85,B 0,C 180,E1 27412.032,E2 27412.032} C_VEL
LIN {X 0,Y 184.775,Z 996.304,A -85,B 0,C 180,E1 27413.88,E2 27413.88} C_VEL
LIN {X 0,Y 177.755,Z 988.987,A -85,B 0,C 180,E1 27415.912,E2 27415.912} C_VEL
LIN {X 0,Y 173.734,Z 977.53,A -85,B 0,C 180,E1 27417.979,E2 27417.979} C_VEL
LIN {X 0,Y 174.674,Z 977.53,A -85,B 0,C 180,E1 27429.672,E2 27429.672} C_VEL
LIN {X 0,Y 175.937,Z 977.53,A -85,B 0,C 180,E1 27440.058,E2 27440.058} C_VEL
LIN {X 0,Y 177.422,Z 977.53,A -85,B 0,C 180,E1 27449.977,E2 27449.977} C_VEL
LIN {X 0,Y 175.911,Z 977.53,A -85,B 0,C 180,E1 27459.897,E2 27459.897} C_VEL
LIN {X 0,Y 175.289,Z 977.951,A -85,B 0,C 180,E1 27465.165,E2 27465.165} C_VEL
LIN {X 0,Y 194.034,Z 1020.491,A -85,B 0,C 180,E1 27474.488,E2 27474.488} C_VEL
LIN {X 0,Y 206.808,Z 1056.398,A -85,B 0,C 180,E1 27480.833,E2 27480.833} C_VEL
LIN {X 0,Y 217.021,Z 1093.844,A -85,B 0,C 180,E1 27487.318,E2 27487.318} C_VEL
LIN {X 0,Y 220.511,Z 1111.605,A -85,B 0,C 180,E1 27490.463,E2 27490.463} C_VEL
LIN {X 0,Y 207.779,Z 1151.605,A -85,B 0,C 180,E1 27496.457,E2 27496.457} C_VEL
LIN {X 0,Y 196.006,Z 1185.46,A -85,B 0,C 180,E1 27503.94,E2 27503.94} C_VEL
LIN {X 0,Y 186.722,Z 1213.642,A -85,B 0,C 180,E1 27512.887,E2 27512.887} C_VEL
LIN {X 0,Y 180.892,Z 1236,A -85,B 0,C 180,E1 27522.918,E2 27522.918} C_VEL
LIN {X 0,Y 178.467,Z 1253.263,A -85,B 0,C 180,E1 27533.874,E2 27533.874} C_VEL
LIN {X 0,Y 178.51,Z 1264,A -85,B 0,C 180,E1 27543.615,E2 27543.615} C_VEL
LIN {X 0,Y 182.628,Z 1273.332,A -85,B 0,C 180,E1 27556.771,E2 27556.771} C_VEL
LIN {X 0,Y 199.427,Z 1278.474,A -85,B 0,C 180,E1 27572.091,E2 27572.091} C_VEL
LIN {X 0,Y 223.801,Z 1278.114,A -85,B 0,C 180,E1 27582.57,E2 27582.57} C_VEL
LIN {X 0,Y 207.81,Z 1281.721,A -85,B 0,C 180,E1 27589.012,E2 27589.012} C_VEL
LIN {X 0,Y 186.02,Z 1284.783,A -85,B 0,C 180,E1 27603.552,E2 27603.552} C_VEL
LIN {X 0,Y 179.563,Z 1283.064,A -85,B 0,C 180,E1 27615.359,E2 27615.359} C_VEL
LIN {X 0,Y 179.366,Z 1277.087,A -85,B 0,C 180,E1 27627.602,E2 27627.602} C_VEL
LIN {X 0,Y 179.786,Z 1270.466,A -85,B 0,C 180,E1 27634.857,E2 27634.857} C_VEL
LIN {X 0,Y 180.639,Z 1256.041,A -85,B 0,C 180,E1 27645.281,E2 27645.281} C_VEL
LIN {X 0,Y 186.873,Z 1253.976,A -85,B 0,C 180,E1 27659.136,E2 27659.136} C_VEL
LIN {X 0,Y 204.825,Z 1246.369,A -85,B 0,C 180,E1 27671.771,E2 27671.771} C_VEL
LIN {X 0,Y 232.352,Z 1233.56,A -85,B 0,C 180,E1 27681.524,E2 27681.524} C_VEL
LIN {X 0,Y 255.955,Z 1221.203,A -85,B 0,C 180,E1 27686.989,E2 27686.989} C_VEL
LIN {X 0,Y 231.641,Z 1228.833,A -85,B 0,C 180,E1 27692.782,E2 27692.782} C_VEL
LIN {X 0,Y 213.169,Z 1231.567,A -85,B 0,C 180,E1 27699.215,E2 27699.215} C_VEL
LIN {X 0,Y 195.312,Z 1229.532,A -85,B 0,C 180,E1 27708.85,E2 27708.85} C_VEL
LIN {X 0,Y 185.003,Z 1222.095,A -85,B 0,C 180,E1 27718.86,E2 27718.86} C_VEL
LIN {X 0,Y 180.724,Z 1208.58,A -85,B 0,C 180,E1 27729.687,E2 27729.687} C_VEL
LIN {X 0,Y 181.376,Z 1191.967,A -85,B 0,C 180,E1 27738.67,E2 27738.67} C_VEL
LIN {X 0,Y 184.773,Z 1168.97,A -85,B 0,C 180,E1 27747.306,E2 27747.306} C_VEL
LIN {X 0,Y 190.119,Z 1141.677,A -85,B 0,C 180,E1 27754.29,E2 27754.29} C_VEL
LIN {X 0,Y 195.937,Z 1110.047,A -85,B 0,C 180,E1 27759.669,E2 27759.669} C_VEL
LIN {X 0,Y 201.225,Z 1070.718,A -85,B 0,C 180,E1 27763.885,E2 27763.885} C_VEL
LIN {X 0,Y 189.879,Z 1024.89,A -85,B 0,C 180,E1 27770.113,E2 27770.113} C_VEL
LIN {X 0,Y 177.755,Z 988.987,A -85,B 0,C 180,E1 27775.912,E2 27775.912} C_VEL
LIN {X 0,Y 169.95,Z 980.24,A -85,B 0,C 180,E1 27778.528,E2 27778.528} C_VEL
LIN {X 0,Y 166.052,Z 977.604,A -85,B 0,C 180,E1 27781.076,E2 27781.076} C_VEL
LIN {X 0,Y 165.936,Z 977.53,A -85,B 0,C 180,E1 27781.578,E2 27781.578} C_VEL
LIN {X 0,Y 166.522,Z 977.53,A -85,B 0,C 180,E1 27788.629,E2 27788.629} C_VEL
LIN {X 0,Y 167.889,Z 977.53,A -85,B 0,C 180,E1 27799.576,E2 27799.576} C_VEL
LIN {X 0,Y 169.488,Z 977.53,A -85,B 0,C 180,E1 27809.976,E2 27809.976} C_VEL
LIN {X 0,Y 167.903,Z 977.53,A -85,B 0,C 180,E1 27820.374,E2 27820.374} C_VEL
LIN {X 0,Y 167.521,Z 977.841,A -85,B 0,C 180,E1 27822.546,E2 27822.546} C_VEL
LIN {X 0,Y 184.342,Z 1015.523,A -85,B 0,C 180,E1 27831.708,E2 27831.708} C_VEL
LIN {X 0,Y 197.264,Z 1050.294,A -85,B 0,C 180,E1 27838.355,E2 27838.355} C_VEL
LIN {X 0,Y 207.341,Z 1086.023,A -85,B 0,C 180,E1 27844.792,E2 27844.792} C_VEL
LIN {X 0,Y 212.913,Z 1113.194,A -85,B 0,C 180,E1 27849.766,E2 27849.766} C_VEL
LIN {X 0,Y 199.993,Z 1152.445,A -85,B 0,C 180,E1 27855.88,E2 27855.88} C_VEL
LIN {X 0,Y 187.948,Z 1186.334,A -85,B 0,C 180,E1 27863.691,E2 27863.691} C_VEL
LIN {X 0,Y 178.275,Z 1215.447,A -85,B 0,C 180,E1 27873.447,E2 27873.447} C_VEL
LIN {X 0,Y 172.449,Z 1238.595,A -85,B 0,C 180,E1 27884.681,E2 27884.681} C_VEL
LIN {X 0,Y 170.542,Z 1253.549,A -85,B 0,C 180,E1 27894.867,E2 27894.867} C_VEL
LIN {X 0,Y 170.781,Z 1264.267,A -85,B 0,C 180,E1 27905.053,E2 27905.053} C_VEL
LIN {X 0,Y 176.805,Z 1274.283,A -85,B 0,C 180,E1 27920.008,E2 27920.008} C_VEL
LIN {X 0,Y 192.779,Z 1278.951,A -85,B 0,C 180,E1 27933.338,E2 27933.338} C_VEL
LIN {X 0,Y 213.214,Z 1279.487,A -85,B 0,C 180,E1 27942.344,E2 27942.344} C_VEL
LIN {X 0,Y 210.779,Z 1280.173,A -85,B 0,C 180,E1 27944.065,E2 27944.065} C_VEL
LIN {X 0,Y 187.056,Z 1283.696,A -85,B 0,C 180,E1 27955.482,E2 27955.482} C_VEL
LIN {X 0,Y 173.777,Z 1283.191,A -85,B 0,C 180,E1 27969.612,E2 27969.612} C_VEL
LIN {X 0,Y 171.068,Z 1278.571,A -85,B 0,C 180,E1 27982.389,E2 27982.389} C_VEL
LIN {X 0,Y 172.052,Z 1272.345,A -85,B 0,C 180,E1 27991.285,E2 27991.285} C_VEL
LIN {X 0,Y 172.136,Z 1262.178,A -85,B 0,C 180,E1 28000.164,E2 28000.164} C_VEL
LIN {X 0,Y 172.933,Z 1254.387,A -85,B 0,C 180,E1 28005.614,E2 28005.614} C_VEL
LIN {X 0,Y 179.87,Z 1252.921,A -85,B 0,C 180,E1 28020.387,E2 28020.387} C_VEL
LIN {X 0,Y 198.907,Z 1246.043,A -85,B 0,C 180,E1 28033.312,E2 28033.312} C_VEL
LIN {X 0,Y 229.431,Z 1233.236,A -85,B 0,C 180,E1 28043.569,E2 28043.569} C_VEL
LIN {X 0,Y 242.832,Z 1227.008,A -85,B 0,C 180,E1 28046.552,E2 28046.552} C_VEL
LIN {X 0,Y 243.813,Z 1226.35,A -85,B 0,C 180,E1 28047.179,E2 28047.179} C_VEL
LIN {X 0,Y 221.373,Z 1231.677,A -85,B 0,C 180,E1 28052.891,E2 28052.891} C_VEL
LIN {X 0,Y 205.78,Z 1233.035,A -85,B 0,C 180,E1 28058.432,E2 28058.432} C_VEL
LIN {X 0,Y 187.451,Z 1230.006,A -85,B 0,C 180,E1 28068.376,E2 28068.376} C_VEL
LIN {X 0,Y 176.988,Z 1221.726,A -85,B 0,C 180,E1 28078.809,E2 28078.809} C_VEL
LIN {X 0,Y 172.786,Z 1207.359,A -85,B 0,C 180,E1 28090.137,E2 28090.137} C_VEL
LIN {X 0,Y 173.939,Z 1187.824,A -85,B 0,C 180,E1 28100.428,E2 28100.428} C_VEL
LIN {X 0,Y 177.772,Z 1163.933,A -85,B 0,C 180,E1 28109.034,E2 28109.034} C_VEL
LIN {X 0,Y 183.254,Z 1136.728,A -85,B 0,C 180,E1 28115.767,E2 28115.767} C_VEL
LIN {X 0,Y 189.375,Z 1103.777,A -85,B 0,C 180,E1 28121.12,E2 28121.12} C_VEL
LIN {X 0,Y 193.393,Z 1070.607,A -85,B 0,C 180,E1 28124.731,E2 28124.731} C_VEL
LIN {X 0,Y 182.52,Z 1026.266,A -85,B 0,C 180,E1 28131.081,E2 28131.081} C_VEL
LIN {X 0,Y 169.153,Z 986.808,A -85,B 0,C 180,E1 28137.909,E2 28137.909} C_VEL
LIN {X 0,Y 165.878,Z 977.53,A -85,B 0,C 180,E1 28139.863,E2 28139.863} C_VEL
LIN {X 0,Y 165.936,Z 977.53,A -85,B 0,C 180,E1 28141.578,E2 28141.578} C_VEL
LIN {X 0,Y 163.782,Z 977.53,A -85,B 0,C 180,E1 28146.064,E2 28146.064} C_VEL
LIN {X 0,Y 159.079,Z 977.53,A -85,B 0,C 180,E1 28153.779,E2 28153.779} C_VEL
LIN {X 0,Y 160.676,Z 977.53,A -85,B 0,C 180,E1 28164.563,E2 28164.563} C_VEL
LIN {X 0,Y 161.569,Z 977.53,A -85,B 0,C 180,E1 28169.975,E2 28169.975} C_VEL
LIN {X 0,Y 160.059,Z 977.871,A -85,B 0,C 180,E1 28179.762,E2 28179.762} C_VEL
LIN {X 0,Y 175.953,Z 1013.506,A -85,B 0,C 180,E1 28189.28,E2 28189.28} C_VEL
LIN {X 0,Y 189.1,Z 1048.365,A -85,B 0,C 180,E1 28196.446,E2 28196.446} C_VEL
LIN {X 0,Y 199.602,Z 1085.382,A -85,B 0,C 180,E1 28203.462,E2 28203.462} C_VEL
LIN {X 0,Y 205.692,Z 1113.33,A -85,B 0,C 180,E1 28208.844,E2 28208.844} C_VEL
LIN {X 0,Y 192.698,Z 1151.96,A -85,B 0,C 180,E1 28215.019,E2 28215.019} C_VEL
LIN {X 0,Y 180.46,Z 1185.496,A -85,B 0,C 180,E1 28222.951,E2 28222.951} C_VEL
LIN {X 0,Y 170.721,Z 1213.962,A -85,B 0,C 180,E1 28232.75,E2 28232.75} C_VEL
LIN {X 0,Y 164.617,Z 1237.781,A -85,B 0,C 180,E1 28244.576,E2 28244.576} C_VEL
LIN {X 0,Y 162.657,Z 1253.775,A -85,B 0,C 180,E1 28255.956,E2 28255.956} C_VEL
LIN {X 0,Y 163.153,Z 1264.463,A -85,B 0,C 180,E1 28266.628,E2 28266.628} C_VEL
LIN {X 0,Y 169.366,Z 1273.919,A -85,B 0,C 180,E1 28280.927,E2 28280.927} C_VEL
LIN {X 0,Y 186.201,Z 1279.217,A -85,B 0,C 180,E1 28294.68,E2 28294.68} C_VEL
LIN {X 0,Y 202.842,Z 1280.372,A -85,B 0,C 180,E1 28302.198,E2 28302.198} C_VEL
LIN {X 0,Y 203.456,Z 1280.533,A -85,B 0,C 180,E1 28303.113,E2 28303.113} C_VEL
LIN {X 0,Y 180.518,Z 1283.166,A -85,B 0,C 180,E1 28314.042,E2 28314.042} C_VEL
LIN {X 0,Y 166.369,Z 1281.982,A -85,B 0,C 180,E1 28328.661,E2 28328.661} C_VEL
LIN {X 0,Y 163.368,Z 1277.033,A -85,B 0,C 180,E1 28342.028,E2 28342.028} C_VEL
LIN {X 0,Y 164.367,Z 1270.469,A -85,B 0,C 180,E1 28351.345,E2 28351.345} C_VEL
LIN {X 0,Y 164.54,Z 1258.2,A -85,B 0,C 180,E1 28361.892,E2 28361.892} C_VEL
LIN {X 0,Y 165.253,Z 1252.633,A -85,B 0,C 180,E1 28365.992,E2 28365.992} C_VEL
LIN {X 0,Y 172.958,Z 1251.783,A -85,B 0,C 180,E1 28381.74,E2 28381.74} C_VEL
LIN {X 0,Y 194.396,Z 1245.164,A -85,B 0,C 180,E1 28395.502,E2 28395.502} C_VEL
LIN {X 0,Y 222.847,Z 1234.568,A -85,B 0,C 180,E1 28404.712,E2 28404.712} C_VEL
LIN {X 0,Y 231.36,Z 1231.051,A -85,B 0,C 180,E1 28406.669,E2 28406.669} C_VEL
LIN {X 0,Y 232.416,Z 1230.46,A -85,B 0,C 180,E1 28407.231,E2 28407.231} C_VEL
LIN {X 0,Y 207.717,Z 1234.229,A -85,B 0,C 180,E1 28414.08,E2 28414.08} C_VEL
LIN {X 0,Y 190.112,Z 1233.448,A -85,B 0,C 180,E1 28421.445,E2 28421.445} C_VEL
LIN {X 0,Y 174.077,Z 1226.951,A -85,B 0,C 180,E1 28432.534,E2 28432.534} C_VEL
LIN {X 0,Y 166.191,Z 1214.737,A -85,B 0,C 180,E1 28444.38,E2 28444.38} C_VEL
LIN {X 0,Y 165.097,Z 1196.652,A -85,B 0,C 180,E1 28456.019,E2 28456.019} C_VEL
LIN {X 0,Y 168.117,Z 1173.926,A -85,B 0,C 180,E1 28465.935,E2 28465.935} C_VEL
LIN {X 0,Y 173.632,Z 1146.038,A -85,B 0,C 180,E1 28474.15,E2 28474.15} C_VEL
LIN {X 0,Y 179.56,Z 1116.064,A -85,B 0,C 180,E1 28480.024,E2 28480.024} C_VEL
LIN {X 0,Y 185.745,Z 1077.823,A -85,B 0,C 180,E1 28484.738,E2 28484.738} C_VEL
LIN {X 0,Y 185.033,Z 1067.805,A -85,B 0,C 180,E1 28486.01,E2 28486.01} C_VEL
LIN {X 0,Y 173.958,Z 1023.49,A -85,B 0,C 180,E1 28492.793,E2 28492.793} C_VEL
LIN {X 0,Y 160.948,Z 986.086,A -85,B 0,C 180,E1 28499.805,E2 28499.805} C_VEL
LIN {X 0,Y 158.066,Z 977.53,A -85,B 0,C 180,E1 28501.73,E2 28501.73} C_VEL
LIN {X 0,Y 159.079,Z 977.53,A -85,B 0,C 180,E1 28513.779,E2 28513.779} C_VEL
LIN {X 0,Y 156.972,Z 977.53,A -85,B 0,C 180,E1 28518.465,E2 28518.465} C_VEL
LIN {X 0,Y 152.859,Z 977.53,A -85,B 0,C 180,E1 28526.532,E2 28526.532} C_VEL
LIN {X 0,Y 153.625,Z 977.53,A -85,B 0,C 180,E1 28529.974,E2 28529.974} C_VEL
LIN {X 0,Y 152.534,Z 977.53,A -85,B 0,C 180,E1 28536.496,E2 28536.496} C_VEL
LIN {X 0,Y 154.705,Z 983.235,A -85,B 0,C 180,E1 28538.308,E2 28538.308} C_VEL
LIN {X 0,Y 168.547,Z 1013.588,A -85,B 0,C 180,E1 28547.132,E2 28547.132} C_VEL
LIN {X 0,Y 180.991,Z 1046.37,A -85,B 0,C 180,E1 28554.371,E2 28554.371} C_VEL
LIN {X 0,Y 191.363,Z 1082.584,A -85,B 0,C 180,E1 28561.616,E2 28561.616} C_VEL
LIN {X 0,Y 198.099,Z 1113.816,A -85,B 0,C 180,E1 28567.894,E2 28567.894} C_VEL
LIN {X 0,Y 185.514,Z 1151.256,A -85,B 0,C 180,E1 28574.063,E2 28574.063} C_VEL
LIN {X 0,Y 172.672,Z 1185.571,A -85,B 0,C 180,E1 28582.458,E2 28582.458} C_VEL
LIN {X 0,Y 162.578,Z 1214.601,A -85,B 0,C 180,E1 28592.937,E2 28592.937} C_VEL
LIN {X 0,Y 156.464,Z 1238.41,A -85,B 0,C 180,E1 28605.464,E2 28605.464} C_VEL
LIN {X 0,Y 154.834,Z 1253.94,A -85,B 0,C 180,E1 28617.156,E2 28617.156} C_VEL
LIN {X 0,Y 155.625,Z 1264.572,A -85,B 0,C 180,E1 28628.357,E2 28628.357} C_VEL
LIN {X 0,Y 164.164,Z 1274.802,A -85,B 0,C 180,E1 28644.497,E2 28644.497} C_VEL
LIN {X 0,Y 187.936,Z 1280.491,A -85,B 0,C 180,E1 28660.118,E2 28660.118} C_VEL
LIN {X 0,Y 193.02,Z 1280.822,A -85,B 0,C 180,E1 28662.221,E2 28662.221} C_VEL
LIN {X 0,Y 193.511,Z 1281.001,A -85,B 0,C 180,E1 28663.079,E2 28663.079} C_VEL
LIN {X 0,Y 167.741,Z 1282.391,A -85,B 0,C 180,E1 28677.209,E2 28677.209} C_VEL
LIN {X 0,Y 156.794,Z 1279.096,A -85,B 0,C 180,E1 28693.174,E2 28693.174} C_VEL
LIN {X 0,Y 156.295,Z 1271.894,A -85,B 0,C 180,E1 28707.247,E2 28707.247} C_VEL
LIN {X 0,Y 156.608,Z 1264.317,A -85,B 0,C 180,E1 28715.578,E2 28715.578} C_VEL
LIN {X 0,Y 157.593,Z 1250.732,A -85,B 0,C 180,E1 28726.115,E2 28726.115} C_VEL
LIN {X 0,Y 166.174,Z 1250.526,A -85,B 0,C 180,E1 28743.198,E2 28743.198} C_VEL
LIN {X 0,Y 187.527,Z 1245.071,A -85,B 0,C 180,E1 28756.685,E2 28756.685} C_VEL
LIN {X 0,Y 218.358,Z 1234.945,A -85,B 0,C 180,E1 28766.413,E2 28766.413} C_VEL
LIN {X 0,Y 220.595,Z 1233.938,A -85,B 0,C 180,E1 28767.372,E2 28767.372} C_VEL
LIN {X 0,Y 200.622,Z 1235.759,A -85,B 0,C 180,E1 28773.091,E2 28773.091} C_VEL
LIN {X 0,Y 178.689,Z 1233.215,A -85,B 0,C 180,E1 28782.773,E2 28782.773} C_VEL
LIN {X 0,Y 164.951,Z 1225.649,A -85,B 0,C 180,E1 28793.445,E2 28793.445} C_VEL
LIN {X 0,Y 157.877,Z 1212.374,A -85,B 0,C 180,E1 28805.546,E2 28805.546} C_VEL
LIN {X 0,Y 157.312,Z 1194.514,A -85,B 0,C 180,E1 28816.835,E2 28816.835} C_VEL
LIN {X 0,Y 160.52,Z 1171.993,A -85,B 0,C 180,E1 28826.7,E2 28826.7} C_VEL
LIN {X 0,Y 165.89,Z 1145.658,A -85,B 0,C 180,E1 28834.665,E2 28834.665} C_VEL
LIN {X 0,Y 172.44,Z 1113.427,A -85,B 0,C 180,E1 28841.101,E2 28841.101} C_VEL
LIN {X 0,Y 178.584,Z 1074.317,A -85,B 0,C 180,E1 28845.983,E2 28845.983} C_VEL
LIN {X 0,Y 168.172,Z 1030.138,A -85,B 0,C 180,E1 28853.018,E2 28853.018} C_VEL
LIN {X 0,Y 156.029,Z 993.638,A -85,B 0,C 180,E1 28860.062,E2 28860.062} C_VEL
LIN {X 0,Y 150.235,Z 977.53,A -85,B 0,C 180,E1 28863.867,E2 28863.867} C_VEL
LIN {X 0,Y 151.028,Z 977.53,A -85,B 0,C 180,E1 28873.833,E2 28873.833} C_VEL
LIN {X 0,Y 152.658,Z 977.53,A -85,B 0,C 180,E1 28884.277,E2 28884.277} C_VEL
LIN {X 0,Y 152.859,Z 977.53,A -85,B 0,C 180,E1 28886.532,E2 28886.532} C_VEL
LIN {X 0,Y 149.346,Z 977.53,A -85,B 0,C 180,E1 28889.001,E2 28889.001} C_VEL
LIN {X 0,Y 145.29,Z 977.53,A -85,B 0,C 180,E1 28891.594,E2 28891.594} C_VEL
LIN {X 0,Y 145.031,Z 977.7,A -85,B 0,C 180,E1 28892.967,E2 28892.967} C_VEL
LIN {X 0,Y 147.234,Z 983.222,A -85,B 0,C 180,E1 28894.954,E2 28894.954} C_VEL
LIN {X 0,Y 161.153,Z 1013.476,A -85,B 0,C 180,E1 28904.765,E2 28904.765} C_VEL
LIN {X 0,Y 173.797,Z 1047.187,A -85,B 0,C 180,E1 28912.736,E2 28912.736} C_VEL
LIN {X 0,Y 183.845,Z 1083.005,A -85,B 0,C 180,E1 28920.294,E2 28920.294} C_VEL
LIN {X 0,Y 190.565,Z 1114.484,A -85,B 0,C 180,E1 28926.924,E2 28926.924} C_VEL
LIN {X 0,Y 178.391,Z 1150.411,A -85,B 0,C 180,E1 28933.041,E2 28933.041} C_VEL
LIN {X 0,Y 165.133,Z 1184.875,A -85,B 0,C 180,E1 28941.706,E2 28941.706} C_VEL
LIN {X 0,Y 154.909,Z 1213.433,A -85,B 0,C 180,E1 28952.366,E2 28952.366} C_VEL
LIN {X 0,Y 148.873,Z 1236.285,A -85,B 0,C 180,E1 28964.705,E2 28964.705} C_VEL
LIN {X 0,Y 147.026,Z 1252.448,A -85,B 0,C 180,E1 28977.004,E2 28977.004} C_VEL
LIN {X 0,Y 147.885,Z 1263.463,A -85,B 0,C 180,E1 28988.798,E2 28988.798} C_VEL
LIN {X 0,Y 156.992,Z 1274.309,A -85,B 0,C 180,E1 29005.696,E2 29005.696} C_VEL
LIN {X 0,Y 181.953,Z 1280.732,A -85,B 0,C 180,E1 29021.725,E2 29021.725} C_VEL
LIN {X 0,Y 183.319,Z 1280.885,A -85,B 0,C 180,E1 29022.295,E2 29022.295} C_VEL
LIN {X 0,Y 182.326,Z 1281.135,A -85,B 0,C 180,E1 29023.553,E2 29023.553} C_VEL
LIN {X 0,Y 161.111,Z 1281.351,A -85,B 0,C 180,E1 29035.676,E2 29035.676} C_VEL
LIN {X 0,Y 149.289,Z 1277.592,A -85,B 0,C 180,E1 29052.301,E2 29052.301} C_VEL
LIN {X 0,Y 148.64,Z 1269.926,A -85,B 0,C 180,E1 29067.106,E2 29067.106} C_VEL
LIN {X 0,Y 148.937,Z 1263.615,A -85,B 0,C 180,E1 29074.403,E2 29074.403} C_VEL
LIN {X 0,Y 149.999,Z 1248.723,A -85,B 0,C 180,E1 29086.499,E2 29086.499} C_VEL
LIN {X 0,Y 159.51,Z 1249.202,A -85,B 0,C 180,E1 29104.779,E2 29104.779} C_VEL
LIN {X 0,Y 182.117,Z 1244.469,A -85,B 0,C 180,E1 29118.522,E2 29118.522} C_VEL
LIN {X 0,Y 209.612,Z 1236.536,A -85,B 0,C 180,E1 29127.306,E2 29127.306} C_VEL
LIN {X 0,Y 183.79,Z 1236.431,A -85,B 0,C 180,E1 29135.695,E2 29135.695} C_VEL
LIN {X 0,Y 165.008,Z 1231.07,A -85,B 0,C 180,E1 29145.9,E2 29145.9} C_VEL
LIN {X 0,Y 152.89,Z 1219.661,A -85,B 0,C 180,E1 29158.621,E2 29158.621} C_VEL
LIN {X 0,Y 149.139,Z 1203.663,A -85,B 0,C 180,E1 29171.023,E2 29171.023} C_VEL
LIN {X 0,Y 150.745,Z 1183.067,A -85,B 0,C 180,E1 29182.186,E2 29182.186} C_VEL
LIN {X 0,Y 155.451,Z 1157.836,A -85,B 0,C 180,E1 29191.639,E2 29191.639} C_VEL
LIN {X 0,Y 161.581,Z 1129.286,A -85,B 0,C 180,E1 29198.883,E2 29198.883} C_VEL
LIN {X 0,Y 168.088,Z 1095.555,A -85,B 0,C 180,E1 29204.355,E2 29204.355} C_VEL
LIN {X 0,Y 170.727,Z 1073.819,A -85,B 0,C 180,E1 29207.041,E2 29207.041} C_VEL
LIN {X 0,Y 160.662,Z 1030.91,A -85,B 0,C 180,E1 29214.267,E2 29214.267} C_VEL
LIN {X 0,Y 148.613,Z 994.337,A -85,B 0,C 180,E1 29221.833,E2 29221.833} C_VEL
LIN {X 0,Y 142.472,Z 977.53,A -85,B 0,C 180,E1 29226.048,E2 29226.048} C_VEL
LIN {X 0,Y 143.655,Z 977.53,A -85,B 0,C 180,E1 29237.793,E2 29237.793} C_VEL
LIN {X 0,Y 144.929,Z 977.53,A -85,B 0,C 180,E1 29246.716,E2 29246.716} C_VEL
LIN {X 0,Y 145.29,Z 977.53,A -85,B 0,C 180,E1 29251.594,E2 29251.594} C_VEL
LIN {X 0,Y 146.402,Z 980.375,A -85,B 0,C 180,E1 29254.041,E2 29254.041} C_VEL
LIN {X 0,Y 148.14,Z 988.235,A -85,B 0,C 180,E1 29256.181,E2 29256.181} C_VEL
LIN {X 0,Y 150.34,Z 1005.453,A -85,B 0,C 180,E1 29259.685,E2 29259.685} C_VEL
LIN {X 0,Y 162.687,Z 1036.186,A -85,B 0,C 180,E1 29268.181,E2 29268.181} C_VEL
LIN {X 0,Y 173.072,Z 1069.851,A -85,B 0,C 180,E1 29275.935,E2 29275.935} C_VEL
LIN {X 0,Y 181.315,Z 1106.068,A -85,B 0,C 180,E1 29283.861,E2 29283.861} C_VEL
LIN {X 0,Y 183.033,Z 1117.292,A -85,B 0,C 180,E1 29286.311,E2 29286.311} C_VEL
LIN {X 0,Y 168.66,Z 1156.124,A -85,B 0,C 180,E1 29293.399,E2 29293.399} C_VEL
LIN {X 0,Y 155.484,Z 1189.712,A -85,B 0,C 180,E1 29302.73,E2 29302.73} C_VEL
LIN {X 0,Y 145.397,Z 1218.083,A -85,B 0,C 180,E1 29314.589,E2 29314.589} C_VEL
LIN {X 0,Y 140.17,Z 1240.397,A -85,B 0,C 180,E1 29328.262,E2 29328.262} C_VEL
LIN {X 0,Y 139.366,Z 1255.602,A -85,B 0,C 180,E1 29341.513,E2 29341.513} C_VEL
LIN {X 0,Y 141.942,Z 1266.607,A -85,B 0,C 180,E1 29355.163,E2 29355.163} C_VEL
LIN {X 0,Y 155.855,Z 1276.403,A -85,B 0,C 180,E1 29372.274,E2 29372.274} C_VEL
LIN {X 0,Y 172.961,Z 1280.452,A -85,B 0,C 180,E1 29382.083,E2 29382.083} C_VEL
LIN {X 0,Y 173.439,Z 1280.709,A -85,B 0,C 180,E1 29383.136,E2 29383.136} C_VEL
LIN {X 0,Y 148.846,Z 1279.332,A -85,B 0,C 180,E1 29399.434,E2 29399.434} C_VEL
LIN {X 0,Y 140.563,Z 1273.274,A -85,B 0,C 180,E1 29417.579,E2 29417.579} C_VEL
LIN {X 0,Y 141.438,Z 1265.572,A -85,B 0,C 180,E1 29430.029,E2 29430.029} C_VEL
LIN {X 0,Y 141.352,Z 1254.197,A -85,B 0,C 180,E1 29440.842,E2 29440.842} C_VEL
LIN {X 0,Y 142.46,Z 1246.575,A -85,B 0,C 180,E1 29446.98,E2 29446.98} C_VEL
LIN {X 0,Y 153.028,Z 1247.754,A -85,B 0,C 180,E1 29466.482,E2 29466.482} C_VEL
LIN {X 0,Y 176.898,Z 1243.704,A -85,B 0,C 180,E1 29480.472,E2 29480.472} C_VEL
LIN {X 0,Y 197.886,Z 1238.569,A -85,B 0,C 180,E1 29487.421,E2 29487.421} C_VEL
LIN {X 0,Y 171.896,Z 1236.349,A -85,B 0,C 180,E1 29496.672,E2 29496.672} C_VEL
LIN {X 0,Y 153.011,Z 1228.228,A -85,B 0,C 180,E1 29508.619,E2 29508.619} C_VEL
LIN {X 0,Y 143.182,Z 1214.611,A -85,B 0,C 180,E1 29522.065,E2 29522.065} C_VEL
LIN {X 0,Y 141.464,Z 1195.798,A -85,B 0,C 180,E1 29535.31,E2 29535.31} C_VEL
LIN {X 0,Y 144.392,Z 1173.456,A -85,B 0,C 180,E1 29546.242,E2 29546.242} C_VEL
LIN {X 0,Y 150.028,Z 1146.477,A -85,B 0,C 180,E1 29555.303,E2 29555.303} C_VEL
LIN {X 0,Y 156.717,Z 1115.567,A -85,B 0,C 180,E1 29562.174,E2 29562.174} C_VEL
LIN {X 0,Y 163.368,Z 1075.905,A -85,B 0,C 180,E1 29567.71,E2 29567.71} C_VEL
LIN {X 0,Y 153.568,Z 1032.874,A -85,B 0,C 180,E1 29575.402,E2 29575.402} C_VEL
LIN {X 0,Y 141.779,Z 996.658,A -85,B 0,C 180,E1 29583.382,E2 29583.382} C_VEL
LIN {X 0,Y 134.618,Z 977.53,A -85,B 0,C 180,E1 29588.51,E2 29588.51} C_VEL
LIN {X 0,Y 135.579,Z 977.53,A -85,B 0,C 180,E1 29597.053,E2 29597.053} C_VEL
LIN {X 0,Y 137.41,Z 977.886,A -85,B 0,C 180,E1 29608.729,E2 29608.729} C_VEL
LIN {X 0,Y 148.535,Z 1001.756,A -85,B 0,C 180,E1 29618.405,E2 29618.405} C_VEL
LIN {X 0,Y 150.34,Z 1005.453,A -85,B 0,C 180,E1 29619.685,E2 29619.685} C_VEL
LIN {X 0,Y 152.733,Z 1016.637,A -85,B 0,C 180,E1 29622.145,E2 29622.145} C_VEL
LIN {X 0,Y 155.447,Z 1036.15,A -85,B 0,C 180,E1 29625.879,E2 29625.879} C_VEL
LIN {X 0,Y 165.851,Z 1070.555,A -85,B 0,C 180,E1 29634.342,E2 29634.342} C_VEL
LIN {X 0,Y 173.927,Z 1107.142,A -85,B 0,C 180,E1 29642.778,E2 29642.778} C_VEL
LIN {X 0,Y 175.786,Z 1117.737,A -85,B 0,C 180,E1 29645.254,E2 29645.254} C_VEL
LIN {X 0,Y 160.958,Z 1156.629,A -85,B 0,C 180,E1 29652.603,E2 29652.603} C_VEL
LIN {X 0,Y 147.074,Z 1191.102,A -85,B 0,C 180,E1 29662.703,E2 29662.703} C_VEL
LIN {X 0,Y 136.929,Z 1219.389,A -85,B 0,C 180,E1 29675.436,E2 29675.436} C_VEL
LIN {X 0,Y 132.209,Z 1240.408,A -85,B 0,C 180,E1 29689.22,E2 29689.22} C_VEL
LIN {X 0,Y 131.735,Z 1255.527,A -85,B 0,C 180,E1 29703.249,E2 29703.249} C_VEL
LIN {X 0,Y 136.1,Z 1267.709,A -85,B 0,C 180,E1 29719.461,E2 29719.461} C_VEL
LIN {X 0,Y 152.904,Z 1277.119,A -85,B 0,C 180,E1 29736.428,E2 29736.428} C_VEL
LIN {X 0,Y 163.779,Z 1279.814,A -85,B 0,C 180,E1 29742.377,E2 29742.377} C_VEL
LIN {X 0,Y 161.867,Z 1279.885,A -85,B 0,C 180,E1 29743.935,E2 29743.935} C_VEL
LIN {X 0,Y 137.443,Z 1276.338,A -85,B 0,C 180,E1 29763.866,E2 29763.866} C_VEL
LIN {X 0,Y 132.854,Z 1269.713,A -85,B 0,C 180,E1 29780.18,E2 29780.18} C_VEL
LIN {X 0,Y 133.807,Z 1263.349,A -85,B 0,C 180,E1 29790.03,E2 29790.03} C_VEL
LIN {X 0,Y 133.779,Z 1250.473,A -85,B 0,C 180,E1 29802.292,E2 29802.292} C_VEL
LIN {X 0,Y 134.943,Z 1244.289,A -85,B 0,C 180,E1 29807.343,E2 29807.343} C_VEL
LIN {X 0,Y 141.084,Z 1246.29,A -85,B 0,C 180,E1 29822.514,E2 29822.514} C_VEL
LIN {X 0,Y 162.294,Z 1244.45,A -85,B 0,C 180,E1 29838.362,E2 29838.362} C_VEL
LIN {X 0,Y 182.548,Z 1240.791,A -85,B 0,C 180,E1 29846.145,E2 29846.145} C_VEL
LIN {X 0,Y 185.559,Z 1239.83,A -85,B 0,C 180,E1 29847.767,E2 29847.767} C_VEL
LIN {X 0,Y 160.041,Z 1235.438,A -85,B 0,C 180,E1 29857.79,E2 29857.79} C_VEL
LIN {X 0,Y 142.307,Z 1225.127,A -85,B 0,C 180,E1 29870.855,E2 29870.855} C_VEL
LIN {X 0,Y 134.352,Z 1209.862,A -85,B 0,C 180,E1 29884.898,E2 29884.898} C_VEL
LIN {X 0,Y 133.97,Z 1190.155,A -85,B 0,C 180,E1 29898.026,E2 29898.026} C_VEL
LIN {X 0,Y 137.549,Z 1167.429,A -85,B 0,C 180,E1 29908.708,E2 29908.708} C_VEL
LIN {X 0,Y 143.993,Z 1138.765,A -85,B 0,C 180,E1 29917.859,E2 29917.859} C_VEL
LIN {X 0,Y 151.138,Z 1105.62,A -85,B 0,C 180,E1 29924.622,E2 29924.622} C_VEL
LIN {X 0,Y 156,Z 1077.82,A -85,B 0,C 180,E1 29928.465,E2 29928.465} C_VEL
LIN {X 0,Y 146.658,Z 1035.573,A -85,B 0,C 180,E1 29936.455,E2 29936.455} C_VEL
LIN {X 0,Y 135.289,Z 999.513,A -85,B 0,C 180,E1 29944.913,E2 29944.913} C_VEL
LIN {X 0,Y 126.88,Z 977.53,A -85,B 0,C 180,E1 29951.579,E2 29951.579} C_VEL
LIN {X 0,Y 128.415,Z 977.981,A -85,B 0,C 180,E1 29962.553,E2 29962.553} C_VEL
LIN {X 0,Y 132.195,Z 983.803,A -85,B 0,C 180,E1 29966.562,E2 29966.562} C_VEL
LIN {X 0,Y 136.218,Z 990.283,A -85,B 0,C 180,E1 29970.364,E2 29970.364} C_VEL
LIN {X 0,Y 148.182,Z 1017.019,A -85,B 0,C 180,E1 29980.467,E2 29980.467} C_VEL
LIN {X 0,Y 155.447,Z 1036.15,A -85,B 0,C 180,E1 29985.879,E2 29985.879} C_VEL
LIN {X 0,Y 157.073,Z 1047.583,A -85,B 0,C 180,E1 29988.159,E2 29988.159} C_VEL
LIN {X 0,Y 157.719,Z 1067.463,A -85,B 0,C 180,E1 29991.708,E2 29991.708} C_VEL
LIN {X 0,Y 165.434,Z 1102.39,A -85,B 0,C 180,E1 30000.221,E2 30000.221} C_VEL
LIN {X 0,Y 168.144,Z 1119.265,A -85,B 0,C 180,E1 30004.295,E2 30004.295} C_VEL
LIN {X 0,Y 152.953,Z 1157.912,A -85,B 0,C 180,E1 30011.959,E2 30011.959} C_VEL
LIN {X 0,Y 139.156,Z 1191.021,A -85,B 0,C 180,E1 30022.178,E2 30022.178} C_VEL
LIN {X 0,Y 128.826,Z 1219.328,A -85,B 0,C 180,E1 30035.64,E2 30035.64} C_VEL
LIN {X 0,Y 124.298,Z 1240.352,A -85,B 0,C 180,E1 30050.301,E2 30050.301} C_VEL
LIN {X 0,Y 124.01,Z 1253.868,A -85,B 0,C 180,E1 30063.452,E2 30063.452} C_VEL
LIN {X 0,Y 129.722,Z 1267.61,A -85,B 0,C 180,E1 30082.256,E2 30082.256} C_VEL
LIN {X 0,Y 153.01,Z 1278.37,A -85,B 0,C 180,E1 30101.887,E2 30101.887} C_VEL
LIN {X 0,Y 153.634,Z 1278.701,A -85,B 0,C 180,E1 30103.237,E2 30103.237} C_VEL
LIN {X 0,Y 130.467,Z 1274.558,A -85,B 0,C 180,E1 30122.353,E2 30122.353} C_VEL
LIN {X 0,Y 125.326,Z 1267.603,A -85,B 0,C 180,E1 30139.584,E2 30139.584} C_VEL
LIN {X 0,Y 126.205,Z 1260.981,A -85,B 0,C 180,E1 30150.032,E2 30150.032} C_VEL
LIN {X 0,Y 126.225,Z 1247.513,A -85,B 0,C 180,E1 30163.041,E2 30163.041} C_VEL
LIN {X 0,Y 127.488,Z 1241.89,A -85,B 0,C 180,E1 30167.91,E2 30167.91} C_VEL
LIN {X 0,Y 134.472,Z 1244.408,A -85,B 0,C 180,E1 30184.328,E2 30184.328} C_VEL
LIN {X 0,Y 157.104,Z 1243.201,A -85,B 0,C 180,E1 30200.538,E2 30200.538} C_VEL
LIN {X 0,Y 172.808,Z 1240.97,A -85,B 0,C 180,E1 30206.615,E2 30206.615} C_VEL
LIN {X 0,Y 174.28,Z 1240.415,A -85,B 0,C 180,E1 30207.771,E2 30207.771} C_VEL
LIN {X 0,Y 148.282,Z 1233.743,A -85,B 0,C 180,E1 30219.091,E2 30219.091} C_VEL
LIN {X 0,Y 131.823,Z 1221.182,A -85,B 0,C 180,E1 30233.448,E2 30233.448} C_VEL
LIN {X 0,Y 125.82,Z 1203.467,A -85,B 0,C 180,E1 30248.707,E2 30248.707} C_VEL
LIN {X 0,Y 127.04,Z 1182.164,A -85,B 0,C 180,E1 30261.934,E2 30261.934} C_VEL
LIN {X 0,Y 132.08,Z 1156.163,A -85,B 0,C 180,E1 30273.072,E2 30273.072} C_VEL
LIN {X 0,Y 139.341,Z 1125.012,A -85,B 0,C 180,E1 30281.817,E2 30281.817} C_VEL
LIN {X 0,Y 146.888,Z 1088.668,A -85,B 0,C 180,E1 30288.043,E2 30288.043} C_VEL
LIN {X 0,Y 148.34,Z 1077.919,A -85,B 0,C 180,E1 30289.591,E2 30289.591} C_VEL
LIN {X 0,Y 138.919,Z 1034.998,A -85,B 0,C 180,E1 30298.303,E2 30298.303} C_VEL
LIN {X 0,Y 127.861,Z 999.619,A -85,B 0,C 180,E1 30307.316,E2 30307.316} C_VEL
LIN {X 0,Y 119.437,Z 979.165,A -85,B 0,C 180,E1 30314.609,E2 30314.609} C_VEL
LIN {X 0,Y 124.111,Z 984.4,A -85,B 0,C 180,E1 30320.61,E2 30320.61} C_VEL
LIN {X 0,Y 130.946,Z 994.176,A -85,B 0,C 180,E1 30327.892,E2 30327.892} C_VEL
LIN {X 0,Y 140.966,Z 1016.885,A -85,B 0,C 180,E1 30337.348,E2 30337.348} C_VEL
LIN {X 0,Y 151.531,Z 1045.951,A -85,B 0,C 180,E1 30346.12,E2 30346.12} C_VEL
LIN {X 0,Y 157.719,Z 1067.463,A -85,B 0,C 180,E1 30351.708,E2 30351.708} C_VEL
LIN {X 0,Y 158.474,Z 1075.037,A -85,B 0,C 180,E1 30353.268,E2 30353.268} C_VEL
LIN {X 0,Y 157.049,Z 1096.749,A -85,B 0,C 180,E1 30357.223,E2 30357.223} C_VEL
LIN {X 0,Y 157.323,Z 1098.547,A -85,B 0,C 180,E1 30357.679,E2 30357.679} C_VEL
LIN {X 0,Y 160.599,Z 1120.543,A -85,B 0,C 180,E1 30363.242,E2 30363.242} C_VEL
LIN {X 0,Y 144.983,Z 1159.06,A -85,B 0,C 180,E1 30371.25,E2 30371.25} C_VEL
LIN {X 0,Y 130.482,Z 1192.79,A -85,B 0,C 180,E1 30382.379,E2 30382.379} C_VEL
LIN {X 0,Y 120.772,Z 1219.205,A -85,B 0,C 180,E1 30395.883,E2 30395.883} C_VEL
LIN {X 0,Y 116.512,Z 1239.318,A -85,B 0,C 180,E1 30410.774,E2 30410.774} C_VEL
LIN {X 0,Y 116.481,Z 1253.652,A -85,B 0,C 180,E1 30425.545,E2 30425.545} C_VEL
LIN {X 0,Y 123.696,Z 1267.357,A -85,B 0,C 180,E1 30445.329,E2 30445.329} C_VEL
LIN {X 0,Y 144.662,Z 1277.112,A -85,B 0,C 180,E1 30462.884,E2 30462.884} C_VEL
LIN {X 0,Y 121.575,Z 1271.569,A -85,B 0,C 180,E1 30484.174,E2 30484.174} C_VEL
LIN {X 0,Y 118.065,Z 1262.277,A -85,B 0,C 180,E1 30504.511,E2 30504.511} C_VEL
LIN {X 0,Y 118.508,Z 1256.941,A -85,B 0,C 180,E1 30511.866,E2 30511.866} C_VEL
LIN {X 0,Y 120.117,Z 1239.332,A -85,B 0,C 180,E1 30528.637,E2 30528.637} C_VEL
LIN {X 0,Y 128.047,Z 1242.42,A -85,B 0,C 180,E1 30546.315,E2 30546.315} C_VEL
LIN {X 0,Y 155.459,Z 1241.536,A -85,B 0,C 180,E1 30564.264,E2 30564.264} C_VEL
LIN {X 0,Y 162.707,Z 1240.745,A -85,B 0,C 180,E1 30566.991,E2 30566.991} C_VEL
LIN {X 0,Y 155.079,Z 1238.578,A -85,B 0,C 180,E1 30570.804,E2 30570.804} C_VEL
LIN {X 0,Y 132.833,Z 1228.826,A -85,B 0,C 180,E1 30583.481,E2 30583.481} C_VEL
LIN {X 0,Y 120.475,Z 1213.475,A -85,B 0,C 180,E1 30599.117,E2 30599.117} C_VEL
LIN {X 0,Y 117.889,Z 1194.569,A -85,B 0,C 180,E1 30613.998,E2 30613.998} C_VEL
LIN {X 0,Y 120.827,Z 1171.688,A -85,B 0,C 180,E1 30626.885,E2 30626.885} C_VEL
LIN {X 0,Y 126.989,Z 1144.43,A -85,B 0,C 180,E1 30637.349,E2 30637.349} C_VEL
LIN {X 0,Y 134.638,Z 1112.008,A -85,B 0,C 180,E1 30645.328,E2 30645.328} C_VEL
LIN {X 0,Y 140.753,Z 1078.404,A -85,B 0,C 180,E1 30650.731,E2 30650.731} C_VEL
LIN {X 0,Y 132.286,Z 1038.34,A -85,B 0,C 180,E1 30659.415,E2 30659.415} C_VEL
LIN {X 0,Y 121.688,Z 1003.094,A -85,B 0,C 180,E1 30668.987,E2 30668.987} C_VEL
LIN {X 0,Y 116.532,Z 988.56,A -85,B 0,C 180,E1 30674.408,E2 30674.408} C_VEL
LIN {X 0,Y 118.873,Z 989.996,A -85,B 0,C 180,E1 30677.301,E2 30677.301} C_VEL
LIN {X 0,Y 122.247,Z 993.58,A -85,B 0,C 180,E1 30681.366,E2 30681.366} C_VEL
LIN {X 0,Y 127.628,Z 1001.454,A -85,B 0,C 180,E1 30687.211,E2 30687.211} C_VEL
LIN {X 0,Y 138.321,Z 1027.627,A -85,B 0,C 180,E1 30697.918,E2 30697.918} C_VEL
LIN {X 0,Y 147.894,Z 1057.982,A -85,B 0,C 180,E1 30707.023,E2 30707.023} C_VEL
LIN {X 0,Y 155.331,Z 1089.132,A -85,B 0,C 180,E1 30715.235,E2 30715.235} C_VEL
LIN {X 0,Y 157.323,Z 1098.547,A -85,B 0,C 180,E1 30717.679,E2 30717.679} C_VEL
LIN {X 0,Y 156.978,Z 1110.069,A -85,B 0,C 180,E1 30720.128,E2 30720.128} C_VEL
LIN {X 0,Y 150.052,Z 1129.437,A -85,B 0,C 180,E1 30723.468,E2 30723.468} C_VEL
LIN {X 0,Y 133.698,Z 1167.294,A -85,B 0,C 180,E1 30732.531,E2 30732.531} C_VEL
LIN {X 0,Y 120.355,Z 1197.868,A -85,B 0,C 180,E1 30744.236,E2 30744.236} C_VEL
LIN {X 0,Y 111.46,Z 1223.093,A -85,B 0,C 180,E1 30759.035,E2 30759.035} C_VEL
LIN {X 0,Y 108.437,Z 1240.947,A -85,B 0,C 180,E1 30773.927,E2 30773.927} C_VEL
LIN {X 0,Y 109.063,Z 1253.338,A -85,B 0,C 180,E1 30787.928,E2 30787.928} C_VEL
LIN {X 0,Y 119.519,Z 1268.072,A -85,B 0,C 180,E1 30810.408,E2 30810.408} C_VEL
LIN {X 0,Y 134.587,Z 1274.934,A -85,B 0,C 180,E1 30822.426,E2 30822.426} C_VEL
LIN {X 0,Y 120.056,Z 1272.035,A -85,B 0,C 180,E1 30834.855,E2 30834.855} C_VEL
LIN {X 0,Y 110.441,Z 1263.033,A -85,B 0,C 180,E1 30858.161,E2 30858.161} C_VEL
LIN {X 0,Y 111.063,Z 1255.903,A -85,B 0,C 180,E1 30870.036,E2 30870.036} C_VEL
LIN {X 0,Y 111.519,Z 1240.139,A -85,B 0,C 180,E1 30885.806,E2 30885.806} C_VEL
LIN {X 0,Y 112.801,Z 1236.672,A -85,B 0,C 180,E1 30889.437,E2 30889.437} C_VEL
LIN {X 0,Y 121.809,Z 1240.284,A -85,B 0,C 180,E1 30908.503,E2 30908.503} C_VEL
LIN {X 0,Y 152.254,Z 1239.804,A -85,B 0,C 180,E1 30927.597,E2 30927.597} C_VEL
LIN {X 0,Y 129.067,Z 1230.554,A -85,B 0,C 180,E1 30939.432,E2 30939.432} C_VEL
LIN {X 0,Y 114.065,Z 1215.165,A -85,B 0,C 180,E1 30955.704,E2 30955.704} C_VEL
LIN {X 0,Y 110.05,Z 1194.994,A -85,B 0,C 180,E1 30972.722,E2 30972.722} C_VEL
LIN {X 0,Y 112.796,Z 1172.01,A -85,B 0,C 180,E1 30986.621,E2 30986.621} C_VEL
LIN {X 0,Y 119.419,Z 1143.239,A -85,B 0,C 180,E1 30998.273,E2 30998.273} C_VEL
LIN {X 0,Y 127.067,Z 1111.872,A -85,B 0,C 180,E1 31006.327,E2 31006.327} C_VEL
LIN {X 0,Y 133.355,Z 1079.963,A -85,B 0,C 180,E1 31011.767,E2 31011.767} C_VEL
LIN {X 0,Y 125.178,Z 1040.049,A -85,B 0,C 180,E1 31021.004,E2 31021.004} C_VEL
LIN {X 0,Y 115.511,Z 1006.384,A -85,B 0,C 180,E1 31030.819,E2 31030.819} C_VEL
LIN {X 0,Y 113.129,Z 998.89,A -85,B 0,C 180,E1 31033.926,E2 31033.926} C_VEL
LIN {X 0,Y 115.895,Z 997.049,A -85,B 0,C 180,E1 31036.38,E2 31036.38} C_VEL
LIN {X 0,Y 119.472,Z 1001.366,A -85,B 0,C 180,E1 31041.014,E2 31041.014} C_VEL
LIN {X 0,Y 123.586,Z 1007.598,A -85,B 0,C 180,E1 31045.762,E2 31045.762} C_VEL
LIN {X 0,Y 132.728,Z 1031.166,A -85,B 0,C 180,E1 31055.908,E2 31055.908} C_VEL
LIN {X 0,Y 141.711,Z 1061.049,A -85,B 0,C 180,E1 31065.47,E2 31065.47} C_VEL
LIN {X 0,Y 148.784,Z 1093.052,A -85,B 0,C 180,E1 31074.408,E2 31074.408} C_VEL
LIN {X 0,Y 153.465,Z 1120.821,A -85,B 0,C 180,E1 31081.947,E2 31081.947} C_VEL
LIN {X 0,Y 150.052,Z 1129.437,A -85,B 0,C 180,E1 31083.468,E2 31083.468} C_VEL
LIN {X 0,Y 140.59,Z 1143.24,A -85,B 0,C 180,E1 31085.571,E2 31085.571} C_VEL
LIN {X 0,Y 131.094,Z 1156.519,A -85,B 0,C 180,E1 31088.301,E2 31088.301} C_VEL
LIN {X 0,Y 115.698,Z 1190.076,A -85,B 0,C 180,E1 31100.132,E2 31100.132} C_VEL
LIN {X 0,Y 104.612,Z 1218.677,A -85,B 0,C 180,E1 31116.465,E2 31116.465} C_VEL
LIN {X 0,Y 100.816,Z 1238.456,A -85,B 0,C 180,E1 31133.466,E2 31133.466} C_VEL
LIN {X 0,Y 101.521,Z 1251.311,A -85,B 0,C 180,E1 31148.521,E2 31148.521} C_VEL
LIN {X 0,Y 111.286,Z 1265.613,A -85,B 0,C 180,E1 31170.635,E2 31170.635} C_VEL
LIN {X 0,Y 122.861,Z 1271.68,A -85,B 0,C 180,E1 31181.001,E2 31181.001} C_VEL
LIN {X 0,Y 124.797,Z 1272.611,A -85,B 0,C 180,E1 31183.286,E2 31183.286} C_VEL
LIN {X 0,Y 104.464,Z 1264.351,A -85,B 0,C 180,E1 31208.78,E2 31208.78} C_VEL
LIN {X 0,Y 103.645,Z 1254.693,A -85,B 0,C 180,E1 31227.944,E2 31227.944} C_VEL
LIN {X 0,Y 103.339,Z 1241.357,A -85,B 0,C 180,E1 31242.746,E2 31242.746} C_VEL
LIN {X 0,Y 105.565,Z 1233.803,A -85,B 0,C 180,E1 31250.092,E2 31250.092} C_VEL
LIN {X 0,Y 115.815,Z 1238.009,A -85,B 0,C 180,E1 31270.903,E2 31270.903} C_VEL
LIN {X 0,Y 141.209,Z 1238.547,A -85,B 0,C 180,E1 31287.609,E2 31287.609} C_VEL
LIN {X 0,Y 117.548,Z 1226.812,A -85,B 0,C 180,E1 31301.258,E2 31301.258} C_VEL
LIN {X 0,Y 104.798,Z 1210.197,A -85,B 0,C 180,E1 31318.379,E2 31318.379} C_VEL
LIN {X 0,Y 102.442,Z 1188.995,A -85,B 0,C 180,E1 31335.903,E2 31335.903} C_VEL
LIN {X 0,Y 106.35,Z 1164.291,A -85,B 0,C 180,E1 31350.304,E2 31350.304} C_VEL
LIN {X 0,Y 113.552,Z 1135.798,A -85,B 0,C 180,E1 31361.281,E2 31361.281} C_VEL
LIN {X 0,Y 121.714,Z 1102.53,A -85,B 0,C 180,E1 31369.241,E2 31369.241} C_VEL
LIN {X 0,Y 125.868,Z 1081.054,A -85,B 0,C 180,E1 31372.952,E2 31372.952} C_VEL
LIN {X 0,Y 118.257,Z 1042.029,A -85,B 0,C 180,E1 31382.697,E2 31382.697} C_VEL
LIN {X 0,Y 109.465,Z 1009.329,A -85,B 0,C 180,E1 31393.114,E2 31393.114} C_VEL
LIN {X 0,Y 114.197,Z 1005.301,A -85,B 0,C 180,E1 31397.128,E2 31397.128} C_VEL
LIN {X 0,Y 119.575,Z 1013.498,A -85,B 0,C 180,E1 31404.112,E2 31404.112} C_VEL
LIN {X 0,Y 128.057,Z 1036.93,A -85,B 0,C 180,E1 31414.618,E2 31414.618} C_VEL
LIN {X 0,Y 135.751,Z 1065.208,A -85,B 0,C 180,E1 31424.178,E2 31424.178} C_VEL
LIN {X 0,Y 142.091,Z 1096.107,A -85,B 0,C 180,E1 31433.271,E2 31433.271} C_VEL
LIN {X 0,Y 145.964,Z 1122.129,A -85,B 0,C 180,E1 31440.737,E2 31440.737} C_VEL
LIN {X 0,Y 131.094,Z 1156.519,A -85,B 0,C 180,E1 31448.301,E2 31448.301} C_VEL
LIN {X 0,Y 124.222,Z 1166.306,A -85,B 0,C 180,E1 31450.805,E2 31450.805} C_VEL
LIN {X 0,Y 112.563,Z 1179.827,A -85,B 0,C 180,E1 31454.972,E2 31454.972} C_VEL
LIN {X 0,Y 111.761,Z 1181.417,A -85,B 0,C 180,E1 31455.617,E2 31455.617} C_VEL
LIN {X 0,Y 99.13,Z 1210.791,A -85,B 0,C 180,E1 31471.399,E2 31471.399} C_VEL
LIN {X 0,Y 93.434,Z 1233.681,A -85,B 0,C 180,E1 31490.601,E2 31490.601} C_VEL
LIN {X 0,Y 93.698,Z 1247.563,A -85,B 0,C 180,E1 31506.899,E2 31506.899} C_VEL
LIN {X 0,Y 103.116,Z 1262.834,A -85,B 0,C 180,E1 31530.878,E2 31530.878} C_VEL
LIN {X 0,Y 115.303,Z 1269.668,A -85,B 0,C 180,E1 31542.294,E2 31542.294} C_VEL
LIN {X 0,Y 113.649,Z 1269.456,A -85,B 0,C 180,E1 31544.817,E2 31544.817} C_VEL
LIN {X 0,Y 96.344,Z 1260.04,A -85,B 0,C 180,E1 31571.71,E2 31571.71} C_VEL
LIN {X 0,Y 96.205,Z 1251.827,A -85,B 0,C 180,E1 31587.785,E2 31587.785} C_VEL
LIN {X 0,Y 96.093,Z 1236.851,A -85,B 0,C 180,E1 31604.891,E2 31604.891} C_VEL
LIN {X 0,Y 98.453,Z 1230.843,A -85,B 0,C 180,E1 31611.243,E2 31611.243} C_VEL
LIN {X 0,Y 110.078,Z 1235.607,A -85,B 0,C 180,E1 31633.544,E2 31633.544} C_VEL
LIN {X 0,Y 128.079,Z 1236.848,A -85,B 0,C 180,E1 31645.965,E2 31645.965} C_VEL
LIN {X 0,Y 129.488,Z 1236.357,A -85,B 0,C 180,E1 31647.859,E2 31647.859} C_VEL
LIN {X 0,Y 108.076,Z 1223.937,A -85,B 0,C 180,E1 31661.674,E2 31661.674} C_VEL
LIN {X 0,Y 95.89,Z 1204.844,A -85,B 0,C 180,E1 31681.196,E2 31681.196} C_VEL
LIN {X 0,Y 95.004,Z 1183.603,A -85,B 0,C 180,E1 31698.668,E2 31698.668} C_VEL
LIN {X 0,Y 99.874,Z 1157.759,A -85,B 0,C 180,E1 31713.485,E2 31713.485} C_VEL
LIN {X 0,Y 107.509,Z 1129.054,A -85,B 0,C 180,E1 31724.173,E2 31724.173} C_VEL
LIN {X 0,Y 116.601,Z 1092.466,A -85,B 0,C 180,E1 31732.408,E2 31732.408} C_VEL
LIN {X 0,Y 118.237,Z 1080.469,A -85,B 0,C 180,E1 31734.689,E2 31734.689} C_VEL
LIN {X 0,Y 111.201,Z 1043.211,A -85,B 0,C 180,E1 31744.757,E2 31744.757} C_VEL
LIN {X 0,Y 105.97,Z 1020.3,A -85,B 0,C 180,E1 31752.674,E2 31752.674} C_VEL
LIN {X 0,Y 112.379,Z 1013.982,A -85,B 0,C 180,E1 31757.887,E2 31757.887} C_VEL
LIN {X 0,Y 116.067,Z 1020.746,A -85,B 0,C 180,E1 31763.107,E2 31763.107} C_VEL
LIN {X 0,Y 123.063,Z 1042.068,A -85,B 0,C 180,E1 31773.048,E2 31773.048} C_VEL
LIN {X 0,Y 130.338,Z 1071.26,A -85,B 0,C 180,E1 31783.413,E2 31783.413} C_VEL
LIN {X 0,Y 136.089,Z 1103.06,A -85,B 0,C 180,E1 31793.337,E2 31793.337} C_VEL
LIN {X 0,Y 138.595,Z 1123.162,A -85,B 0,C 180,E1 31799.384,E2 31799.384} C_VEL
LIN {X 0,Y 121.242,Z 1161.396,A -85,B 0,C 180,E1 31808.431,E2 31808.431} C_VEL
LIN {X 0,Y 111.761,Z 1181.417,A -85,B 0,C 180,E1 31815.617,E2 31815.617} C_VEL
LIN {X 0,Y 105.234,Z 1190.338,A -85,B 0,C 180,E1 31819.355,E2 31819.355} C_VEL
LIN {X 0,Y 94.302,Z 1202.422,A -85,B 0,C 180,E1 31825.929,E2 31825.929} C_VEL
LIN {X 0,Y 93.608,Z 1203.834,A -85,B 0,C 180,E1 31826.872,E2 31826.872} C_VEL
LIN {X 0,Y 86.145,Z 1228.55,A -85,B 0,C 180,E1 31847.367,E2 31847.367} C_VEL
LIN {X 0,Y 85.891,Z 1243.422,A -85,B 0,C 180,E1 31864.988,E2 31864.988} C_VEL
LIN {X 0,Y 93.578,Z 1258.569,A -85,B 0,C 180,E1 31888.984,E2 31888.984} C_VEL
LIN {X 0,Y 106.269,Z 1266.658,A -85,B 0,C 180,E1 31902.587,E2 31902.587} C_VEL
LIN {X 0,Y 105.537,Z 1266.615,A -85,B 0,C 180,E1 31904.175,E2 31904.175} C_VEL
LIN {X 0,Y 88.857,Z 1256.296,A -85,B 0,C 180,E1 31932.762,E2 31932.762} C_VEL
LIN {X 0,Y 88.752,Z 1248.934,A -85,B 0,C 180,E1 31947.599,E2 31947.599} C_VEL
LIN {X 0,Y 89.23,Z 1232.09,A -85,B 0,C 180,E1 31967.335,E2 31967.335} C_VEL
LIN {X 0,Y 91.377,Z 1227.634,A -85,B 0,C 180,E1 31972.079,E2 31972.079} C_VEL
LIN {X 0,Y 104.633,Z 1233.084,A -85,B 0,C 180,E1 31996.449,E2 31996.449} C_VEL
LIN {X 0,Y 116.404,Z 1234.31,A -85,B 0,C 180,E1 32005.043,E2 32005.043} C_VEL
LIN {X 0,Y 118.909,Z 1233.978,A -85,B 0,C 180,E1 32007.668,E2 32007.668} C_VEL
LIN {X 0,Y 96.864,Z 1218.679,A -85,B 0,C 180,E1 32024.18,E2 32024.18} C_VEL
LIN {X 0,Y 87.245,Z 1198.288,A -85,B 0,C 180,E1 32045.053,E2 32045.053} C_VEL
LIN {X 0,Y 88.048,Z 1176.222,A -85,B 0,C 180,E1 32062.855,E2 32062.855} C_VEL
LIN {X 0,Y 93.933,Z 1150.121,A -85,B 0,C 180,E1 32077.312,E2 32077.312} C_VEL
LIN {X 0,Y 102.581,Z 1118.546,A -85,B 0,C 180,E1 32088.261,E2 32088.261} C_VEL
LIN {X 0,Y 111.116,Z 1083.381,A -85,B 0,C 180,E1 32095.668,E2 32095.668} C_VEL
LIN {X 0,Y 104.653,Z 1046.16,A -85,B 0,C 180,E1 32106.494,E2 32106.494} C_VEL
LIN {X 0,Y 101.769,Z 1031.752,A -85,B 0,C 180,E1 32111.678,E2 32111.678} C_VEL
LIN {X 0,Y 110.316,Z 1022.822,A -85,B 0,C 180,E1 32118.459,E2 32118.459} C_VEL
LIN {X 0,Y 113.532,Z 1030.989,A -85,B 0,C 180,E1 32123.764,E2 32123.764} C_VEL
LIN {X 0,Y 120.049,Z 1054.83,A -85,B 0,C 180,E1 32134.488,E2 32134.488} C_VEL
LIN {X 0,Y 126.335,Z 1085.928,A -85,B 0,C 180,E1 32145.539,E2 32145.539} C_VEL
LIN {X 0,Y 131.083,Z 1119.895,A -85,B 0,C 180,E1 32156.577,E2 32156.577} C_VEL
LIN {X 0,Y 131.054,Z 1124.472,A -85,B 0,C 180,E1 32157.955,E2 32157.955} C_VEL
LIN {X 0,Y 113.305,Z 1162.25,A -85,B 0,C 180,E1 32167.354,E2 32167.354} C_VEL
